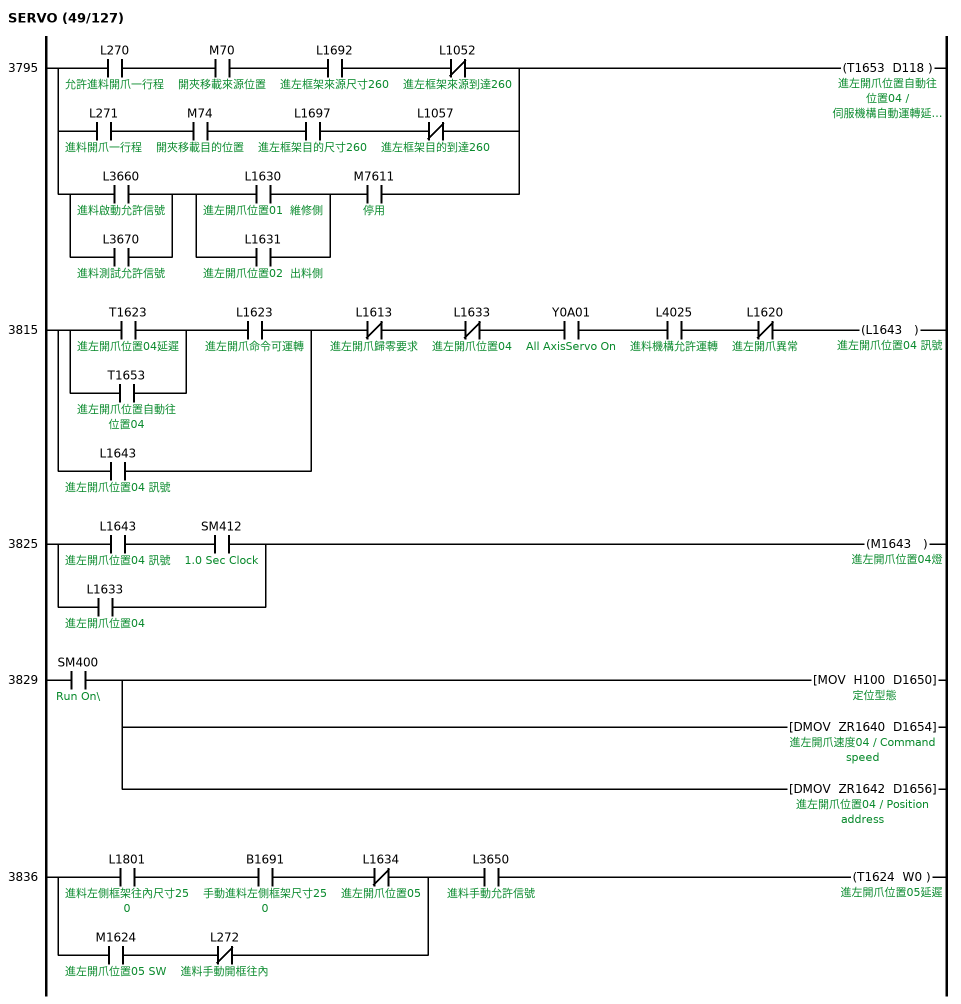
[picture p48: ladder of SERVO, rungs at steps 3795 to 3836]
3795  LD      L270  ; 允許進料開爪一行程
      AND     M70  ; 開夾移載來源位置
      AND     L1692  ; 進左框架來源尺寸260
      ANI     L1052  ; 進左框架來源到達260
      LD      L271  ; 進料開爪一行程
      AND     M74  ; 開夾移載目的位置
      AND     L1697  ; 進左框架目的尺寸260
      ANI     L1057  ; 進左框架目的到達260
      ORB
      LD      L3660  ; 進料啟動允許信號
      OR      L3670  ; 進料測試允許信號
      LD      L1630  ; 進左開爪位置01  維修側
      OR      L1631  ; 進左開爪位置02  出料側
      ANB
      AND     M7611  ; 停用
      ORB
      OUT     T1653 D118  ; 進左開爪位置自動往  位置04 / 伺服機構自動運轉延遲時間
3815  LD      T1623  ; 進左開爪位置04延遲
      OR      T1653  ; 進左開爪位置自動往  位置04
      AND     L1623  ; 進左開爪命令可運轉
      OR      L1643  ; 進左開爪位置04 訊號
      ANI     L1613  ; 進左開爪歸零要求
      ANI     L1633  ; 進左開爪位置04
      AND     Y0A01  ; All AxisServo On
      AND     L4025  ; 進料機構允許運轉
      ANI     L1620  ; 進左開爪異常
      OUT     L1643  ; 進左開爪位置04 訊號
3825  LD      L1643  ; 進左開爪位置04 訊號
      AND     SM412  ; 1.0 Sec Clock
      OR      L1633  ; 進左開爪位置04
      OUT     M1643  ; 進左開爪位置04燈
3829  LD      SM400  ; Run On\
      MOV     H100 D1650  ; 定位型態
      DMOV    ZR1640 D1654  ; 進左開爪速度04 / Command  speed
      DMOV    ZR1642 D1656  ; Position address
3836  LD      L1801  ; 進料左側框架往內尺寸250
      AND     B1691  ; 手動進料左側框架尺寸250
      ANI     L1634  ; 進左開爪位置05
      LD      M1624  ; 進左開爪位置05 SW
      ANI     L272  ; 進料手動開框往內
      ORB
      AND     L3650  ; 進料手動允許信號
      OUT     T1624 W0  ; 進左開爪位置05延遲
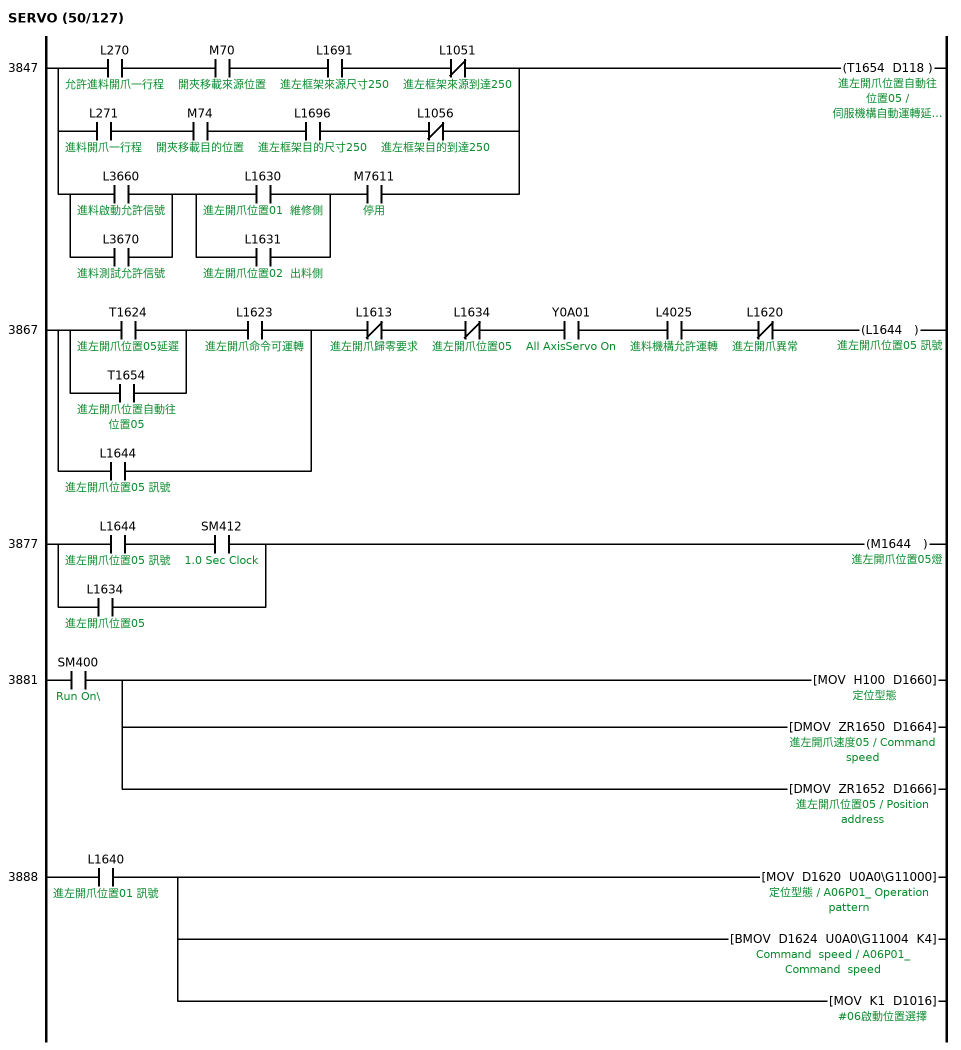
3847  LD      L270  ; 允許進料開爪一行程
      AND     M70  ; 開夾移載來源位置
      AND     L1691  ; 進左框架來源尺寸250
      ANI     L1051  ; 進左框架來源到達250
      LD      L271  ; 進料開爪一行程
      AND     M74  ; 開夾移載目的位置
      AND     L1696  ; 進左框架目的尺寸250
      ANI     L1056  ; 進左框架目的到達250
      ORB
      LD      L3660  ; 進料啟動允許信號
      OR      L3670  ; 進料測試允許信號
      LD      L1630  ; 進左開爪位置01  維修側
      OR      L1631  ; 進左開爪位置02  出料側
      ANB
      AND     M7611  ; 停用
      ORB
      OUT     T1654 D118  ; 進左開爪位置自動往  位置05 / 伺服機構自動運轉延遲時間
3867  LD      T1624  ; 進左開爪位置05延遲
      OR      T1654  ; 進左開爪位置自動往  位置05
      AND     L1623  ; 進左開爪命令可運轉
      OR      L1644  ; 進左開爪位置05 訊號
      ANI     L1613  ; 進左開爪歸零要求
      ANI     L1634  ; 進左開爪位置05
      AND     Y0A01  ; All AxisServo On
      AND     L4025  ; 進料機構允許運轉
      ANI     L1620  ; 進左開爪異常
      OUT     L1644  ; 進左開爪位置05 訊號
3877  LD      L1644  ; 進左開爪位置05 訊號
      AND     SM412  ; 1.0 Sec Clock
      OR      L1634  ; 進左開爪位置05
      OUT     M1644  ; 進左開爪位置05燈
3881  LD      SM400  ; Run On\
      MOV     H100 D1660  ; 定位型態
      DMOV    ZR1650 D1664  ; 進左開爪速度05 / Command  speed
      DMOV    ZR1652 D1666  ; Position address
3888  LD      L1640  ; 進左開爪位置01 訊號
      MOV     D1620 U0A0\G11000  ; A06P01_ Operation pattern
      BMOV    D1624 U0A0\G11004 K4  ; A06P01_ Command  speed
      MOV     K1 D1016  ; #06啟動位置選擇
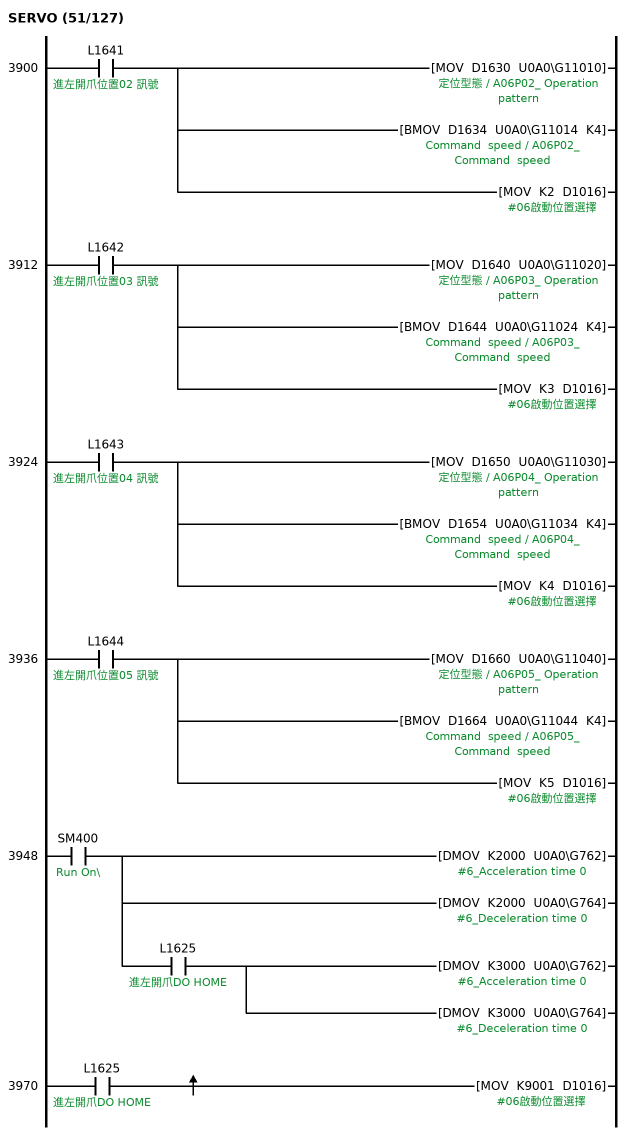
3900  LD      L1641  ; 進左開爪位置02 訊號
      MOV     D1630 U0A0\G11010  ; A06P02_ Operation pattern
      BMOV    D1634 U0A0\G11014 K4  ; A06P02_ Command  speed
      MOV     K2 D1016
3912  LD      L1642  ; 進左開爪位置03 訊號
      MOV     D1640 U0A0\G11020  ; A06P03_ Operation pattern
      BMOV    D1644 U0A0\G11024 K4  ; A06P03_ Command  speed
      MOV     K3 D1016
3924  LD      L1643  ; 進左開爪位置04 訊號
      MOV     D1650 U0A0\G11030  ; A06P04_ Operation pattern
      BMOV    D1654 U0A0\G11034 K4  ; A06P04_ Command  speed
      MOV     K4 D1016
3936  LD      L1644  ; 進左開爪位置05 訊號
      MOV     D1660 U0A0\G11040  ; A06P05_ Operation pattern
      BMOV    D1664 U0A0\G11044 K4  ; A06P05_ Command  speed
      MOV     K5 D1016
3948  LD      SM400  ; Run On\
      DMOV    K2000 U0A0\G762  ; #6_Acceleration time 0
      DMOV    K2000 U0A0\G764  ; #6_Deceleration time 0
      AND     L1625  ; 進左開爪DO HOME
      DMOV    K3000 U0A0\G762
      DMOV    K3000 U0A0\G764
3970  LD      L1625  ; 進左開爪DO HOME
      MEP
      MOV     K9001 D1016
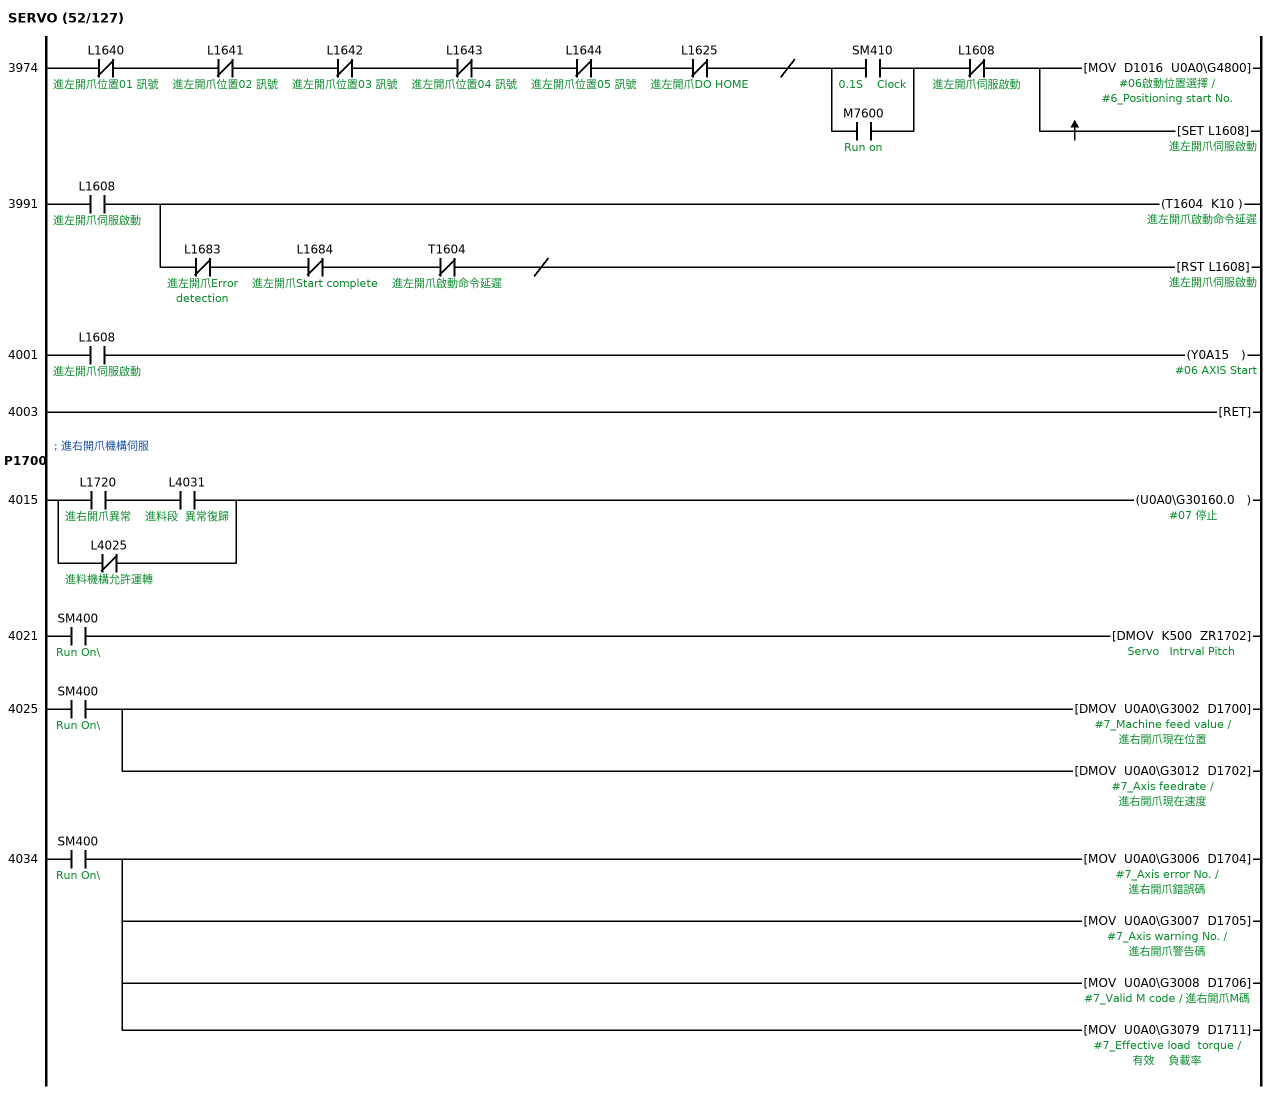
3974  LDI     L1640  ; 進左開爪位置01 訊號
      ANI     L1641  ; 進左開爪位置02 訊號
      ANI     L1642  ; 進左開爪位置03 訊號
      ANI     L1643  ; 進左開爪位置04 訊號
      ANI     L1644  ; 進左開爪位置05 訊號
      ANI     L1625  ; 進左開爪DO HOME
      INV
      LD      SM410  ; 0.1S    Clock
      OR      M7600  ; Run on
      ANB
      ANI     L1608  ; 進左開爪伺服啟動
      MOV     D1016 U0A0\G4800  ; #6_Positioning start No.
      MEP
      SET     L1608  ; 進左開爪伺服啟動
3991  LD      L1608  ; 進左開爪伺服啟動
      OUT     T1604 K10  ; 進左開爪啟動命令延遲
      ANI     L1683  ; 進左開爪Error detection
      ANI     L1684  ; 進左開爪Start complete
      ANI     T1604  ; 進左開爪啟動命令延遲
      INV
      RST     L1608  ; 進左開爪伺服啟動
4001  LD      L1608  ; 進左開爪伺服啟動
      OUT     Y0A15  ; #06 AXIS Start
4003  RET
; 進右開爪機構伺服
      P1700
4015  LD      L1720  ; 進右開爪異常
      AND     L4031  ; 進料段  異常復歸
      ORI     L4025  ; 進料機構允許運轉
      OUT     U0A0\G30160.0  ; #07 停止
4021  LD      SM400  ; Run On\
      DMOV    K500 ZR1702  ; Servo   Intrval Pitch
4025  LD      SM400  ; Run On\
      DMOV    U0A0\G3002 D1700  ; #7_Machine feed value / 進右開爪現在位置
      DMOV    U0A0\G3012 D1702  ; #7_Axis feedrate / 進右開爪現在速度
4034  LD      SM400  ; Run On\
      MOV     U0A0\G3006 D1704  ; #7_Axis error No. / 進右開爪錯誤碼
      MOV     U0A0\G3007 D1705  ; #7_Axis warning No. / 進右開爪警告碼
      MOV     U0A0\G3008 D1706  ; #7_Valid M code / 進右開爪M碼
      MOV     U0A0\G3079 D1711  ; #7_Effective load  torque / 有效    負載率
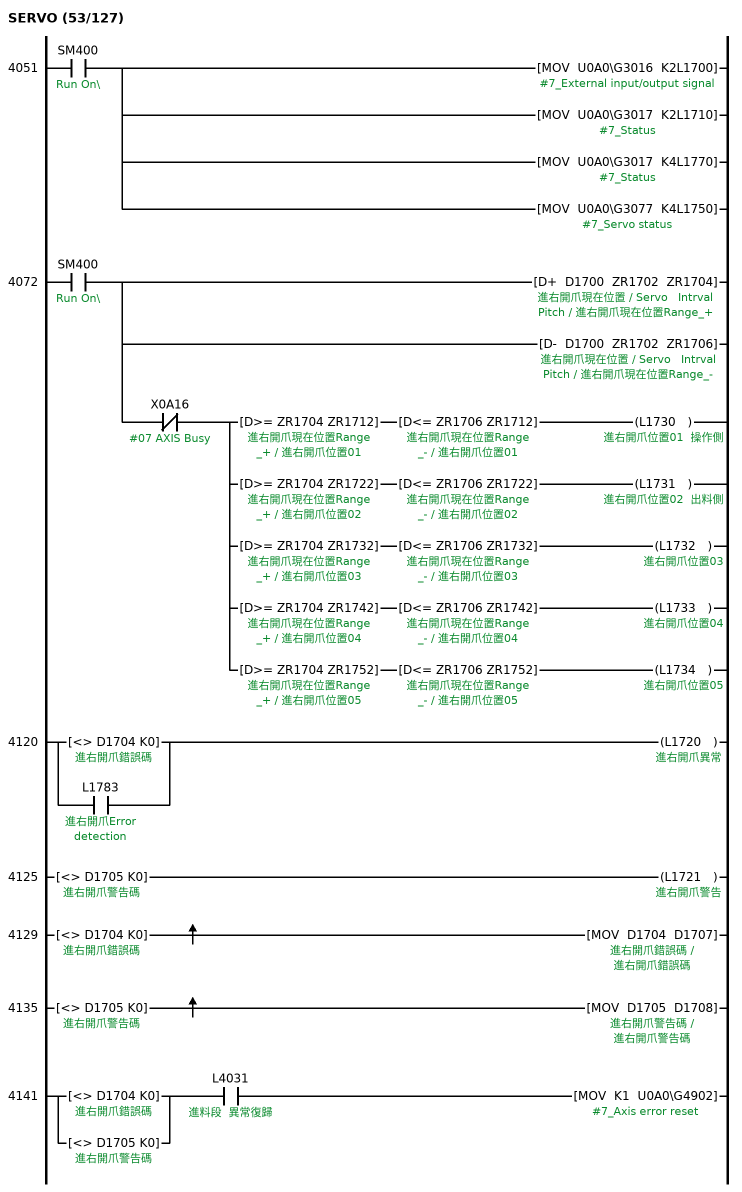
4051  LD      SM400  ; Run On\
      MOV     U0A0\G3016 K2L1700  ; #7_External input/output signal / 進右開爪  負極限
      MOV     U0A0\G3017 K2L1710  ; #7_Status / 進右開爪速度控制
      MOV     U0A0\G3017 K4L1770  ; 進右開爪速度控制
      MOV     U0A0\G3077 K4L1750  ; #7_Servo status / READY ON
4072  LD      SM400  ; Run On\
      D+      D1700 ZR1702 ZR1704  ; 進右開爪現在位置Range_+
      D-      D1700 ZR1702 ZR1706  ; 進右開爪現在位置Range_-
      ANI     X0A16  ; #07 AXIS Busy
      MPS
      ANDD>=  ZR1704 ZR1712  ; 進右開爪現在位置Range_+ / 進右開爪位置01
      ANDD<=  ZR1706 ZR1712  ; 進右開爪現在位置Range_- / 進右開爪位置01
      OUT     L1730  ; 進右開爪位置01  操作側
      MRD
      ANDD>=  ZR1704 ZR1722  ; 進右開爪現在位置Range_+ / 進右開爪位置02
      ANDD<=  ZR1706 ZR1722  ; 進右開爪現在位置Range_- / 進右開爪位置02
      OUT     L1731  ; 進右開爪位置02  出料側
      MRD
      ANDD>=  ZR1704 ZR1732  ; 進右開爪現在位置Range_+ / 進右開爪位置03
      ANDD<=  ZR1706 ZR1732  ; 進右開爪現在位置Range_- / 進右開爪位置03
      OUT     L1732  ; 進右開爪位置03
      MRD
      ANDD>=  ZR1704 ZR1742  ; 進右開爪現在位置Range_+ / 進右開爪位置04
      ANDD<=  ZR1706 ZR1742  ; 進右開爪現在位置Range_- / 進右開爪位置04
      OUT     L1733  ; 進右開爪位置04
      MPP
      ANDD>=  ZR1704 ZR1752  ; 進右開爪現在位置Range_+ / 進右開爪位置05
      ANDD<=  ZR1706 ZR1752  ; 進右開爪現在位置Range_- / 進右開爪位置05
      OUT     L1734  ; 進右開爪位置05
4120  LD<>    D1704 K0  ; 進右開爪錯誤碼
      OR      L1783  ; 進右開爪Error detection
      OUT     L1720  ; 進右開爪異常
4125  LD<>    D1705 K0  ; 進右開爪警告碼
      OUT     L1721  ; 進右開爪警告
4129  LD<>    D1704 K0  ; 進右開爪錯誤碼
      MEP
      MOV     D1704 D1707  ; 進右開爪錯誤碼
4135  LD<>    D1705 K0  ; 進右開爪警告碼
      MEP
      MOV     D1705 D1708  ; 進右開爪警告碼
4141  LD<>    D1704 K0  ; 進右開爪錯誤碼
      OR<>    D1705 K0  ; 進右開爪警告碼
      AND     L4031  ; 進料段  異常復歸
      MOV     K1 U0A0\G4902  ; #7_Axis error reset
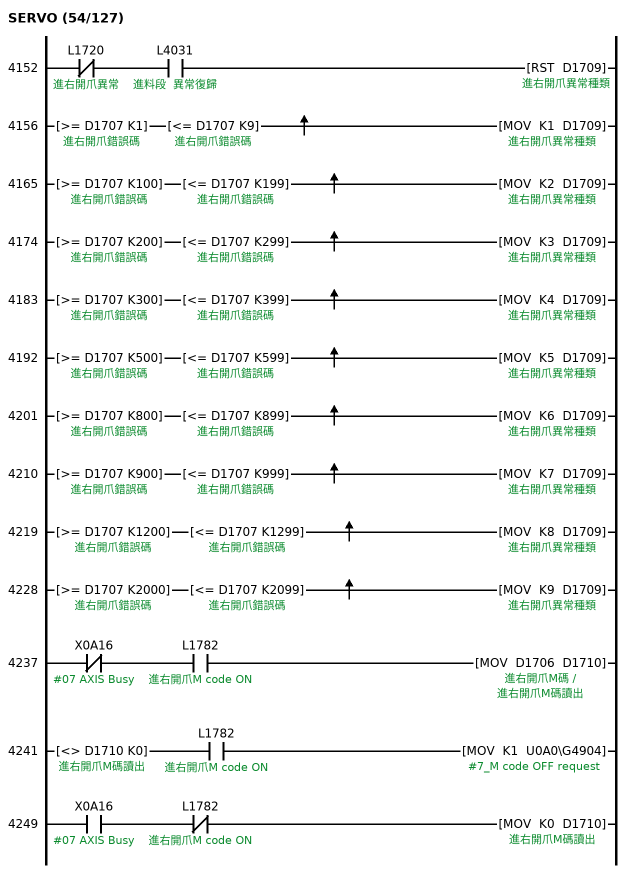
4152  LDI     L1720  ; 進右開爪異常
      AND     L4031  ; 進料段  異常復歸
      RST     D1709  ; 進右開爪異常種類
4156  LD>=    D1707 K1  ; 進右開爪錯誤碼
      AND<=   D1707 K9  ; 進右開爪錯誤碼
      MEP
      MOV     K1 D1709
4165  LD>=    D1707 K100  ; 進右開爪錯誤碼
      AND<=   D1707 K199  ; 進右開爪錯誤碼
      MEP
      MOV     K2 D1709
4174  LD>=    D1707 K200  ; 進右開爪錯誤碼
      AND<=   D1707 K299  ; 進右開爪錯誤碼
      MEP
      MOV     K3 D1709
4183  LD>=    D1707 K300  ; 進右開爪錯誤碼
      AND<=   D1707 K399  ; 進右開爪錯誤碼
      MEP
      MOV     K4 D1709
4192  LD>=    D1707 K500  ; 進右開爪錯誤碼
      AND<=   D1707 K599  ; 進右開爪錯誤碼
      MEP
      MOV     K5 D1709
4201  LD>=    D1707 K800  ; 進右開爪錯誤碼
      AND<=   D1707 K899  ; 進右開爪錯誤碼
      MEP
      MOV     K6 D1709
4210  LD>=    D1707 K900  ; 進右開爪錯誤碼
      AND<=   D1707 K999  ; 進右開爪錯誤碼
      MEP
      MOV     K7 D1709
4219  LD>=    D1707 K1200  ; 進右開爪錯誤碼
      AND<=   D1707 K1299  ; 進右開爪錯誤碼
      MEP
      MOV     K8 D1709
4228  LD>=    D1707 K2000  ; 進右開爪錯誤碼
      AND<=   D1707 K2099  ; 進右開爪錯誤碼
      MEP
      MOV     K9 D1709
4237  LDI     X0A16  ; #07 AXIS Busy
      AND     L1782  ; 進右開爪M code ON
      MOV     D1706 D1710  ; 進右開爪M碼讀出
4241  LD<>    D1710 K0  ; 進右開爪M碼讀出
      AND     L1782  ; 進右開爪M code ON
      MOV     K1 U0A0\G4904  ; #7_M code OFF request
4249  LD      X0A16  ; #07 AXIS Busy
      ANI     L1782  ; 進右開爪M code ON
      MOV     K0 D1710
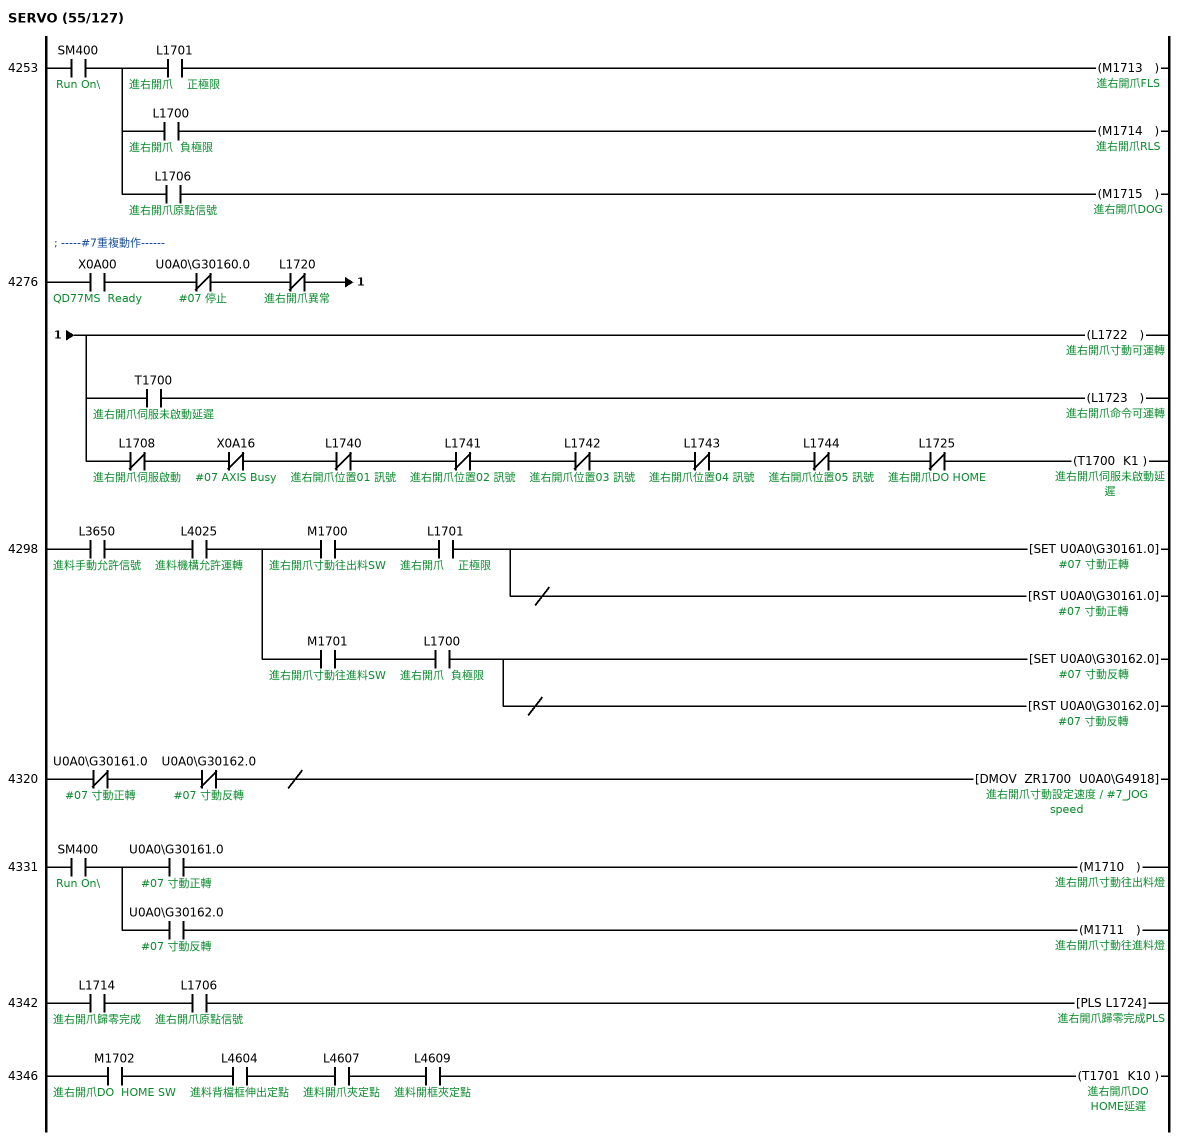
4253  LD      SM400  ; Run On\
      MPS
      AND     L1701  ; 進右開爪    正極限
      OUT     M1713  ; 進右開爪FLS
      MRD
      AND     L1700  ; 進右開爪  負極限
      OUT     M1714  ; 進右開爪RLS
      MPP
      AND     L1706  ; 進右開爪原點信號
      OUT     M1715  ; 進右開爪DOG
; -----#7重複動作------
4276  LD      X0A00  ; QD77MS  Ready
      ANI     U0A0\G30160.0  ; #07 停止
      ANI     L1720  ; 進右開爪異常
      OUT     L1722  ; 進右開爪寸動可運轉
      MPS
      AND     T1700  ; 進右開爪伺服未啟動延遲
      OUT     L1723  ; 進右開爪命令可運轉
      MPP
      ANI     L1708  ; 進右開爪伺服啟動
      ANI     X0A16  ; #07 AXIS Busy
      ANI     L1740  ; 進右開爪位置01 訊號
      ANI     L1741  ; 進右開爪位置02 訊號
      ANI     L1742  ; 進右開爪位置03 訊號
      ANI     L1743  ; 進右開爪位置04 訊號
      ANI     L1744  ; 進右開爪位置05 訊號
      ANI     L1725  ; 進右開爪DO HOME
      OUT     T1700 K1  ; 進右開爪伺服未啟動延遲
4298  LD      L3650  ; 進料手動允許信號
      AND     L4025  ; 進料機構允許運轉
      MPS
      AND     M1700  ; 進右開爪寸動往出料SW
      AND     L1701  ; 進右開爪    正極限
      SET     U0A0\G30161.0  ; #07 寸動正轉
      INV
      RST     U0A0\G30161.0  ; #07 寸動正轉
      MPP
      AND     M1701  ; 進右開爪寸動往進料SW
      AND     L1700  ; 進右開爪  負極限
      SET     U0A0\G30162.0  ; #07 寸動反轉
      INV
      RST     U0A0\G30162.0  ; #07 寸動反轉
4320  LDI     U0A0\G30161.0  ; #07 寸動正轉
      ANI     U0A0\G30162.0  ; #07 寸動反轉
      INV
      DMOV    ZR1700 U0A0\G4918  ; 進右開爪寸動設定速度 / #7_JOG     speed
4331  LD      SM400  ; Run On\
      MPS
      AND     U0A0\G30161.0  ; #07 寸動正轉
      OUT     M1710  ; 進右開爪寸動往出料燈
      MPP
      AND     U0A0\G30162.0  ; #07 寸動反轉
      OUT     M1711  ; 進右開爪寸動往進料燈
4342  LD      L1714  ; 進右開爪歸零完成
      AND     L1706  ; 進右開爪原點信號
      PLS     L1724  ; 進右開爪歸零完成PLS
4346  LD      M1702  ; 進右開爪DO  HOME SW
      AND     L4604  ; 進料背檔框伸出定點
      AND     L4607  ; 進料開爪夾定點
      AND     L4609  ; 進料開框夾定點
      OUT     T1701 K10  ; 進右開爪DO HOME延遲
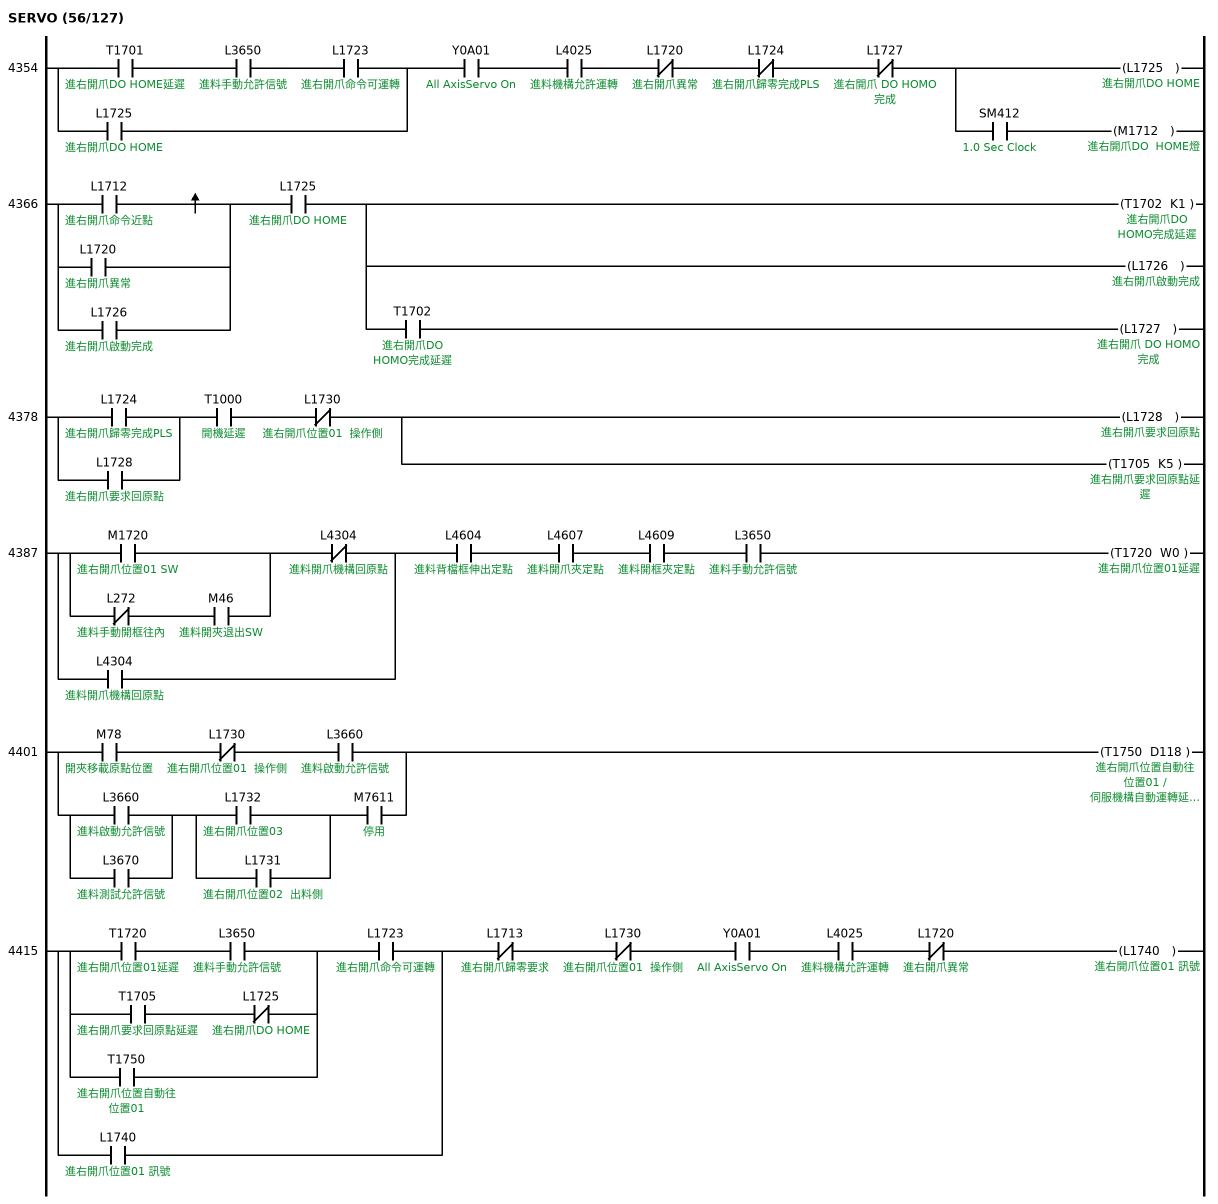
4354  LD      T1701  ; 進右開爪DO HOME延遲
      AND     L3650  ; 進料手動允許信號
      AND     L1723  ; 進右開爪命令可運轉
      OR      L1725  ; 進右開爪DO HOME
      AND     Y0A01  ; All AxisServo On
      AND     L4025  ; 進料機構允許運轉
      ANI     L1720  ; 進右開爪異常
      ANI     L1724  ; 進右開爪歸零完成PLS
      ANI     L1727  ; 進右開爪 DO HOMO 完成
      OUT     L1725  ; 進右開爪DO HOME
      AND     SM412  ; 1.0 Sec Clock
      OUT     M1712  ; 進右開爪DO  HOME燈
4366  LD      L1712  ; 進右開爪命令近點
      MEP
      OR      L1720  ; 進右開爪異常
      OR      L1726  ; 進右開爪啟動完成
      AND     L1725  ; 進右開爪DO HOME
      OUT     T1702 K1  ; 進右開爪DO HOMO完成延遲
      OUT     L1726  ; 進右開爪啟動完成
      AND     T1702  ; 進右開爪DO HOMO完成延遲
      OUT     L1727  ; 進右開爪 DO HOMO 完成
4378  LD      L1724  ; 進右開爪歸零完成PLS
      OR      L1728  ; 進右開爪要求回原點
      AND     T1000  ; 開機延遲
      ANI     L1730  ; 進右開爪位置01  操作側
      OUT     L1728  ; 進右開爪要求回原點
      OUT     T1705 K5  ; 進右開爪要求回原點延遲
4387  LD      M1720  ; 進右開爪位置01 SW
      LDI     L272  ; 進料手動開框往內
      AND     M46  ; 進料開夾退出SW
      ORB
      ANI     L4304  ; 進料開爪機構回原點
      OR      L4304  ; 進料開爪機構回原點
      AND     L4604  ; 進料背檔框伸出定點
      AND     L4607  ; 進料開爪夾定點
      AND     L4609  ; 進料開框夾定點
      AND     L3650  ; 進料手動允許信號
      OUT     T1720 W0  ; 進右開爪位置01延遲
4401  LD      M78  ; 開夾移載原點位置
      ANI     L1730  ; 進右開爪位置01  操作側
      AND     L3660  ; 進料啟動允許信號
      LD      L3660  ; 進料啟動允許信號
      OR      L3670  ; 進料測試允許信號
      LD      L1732  ; 進右開爪位置03
      OR      L1731  ; 進右開爪位置02  出料側
      ANB
      AND     M7611  ; 停用
      ORB
      OUT     T1750 D118  ; 進右開爪位置自動往  位置01 / 伺服機構自動運轉延遲時間
4415  LD      T1720  ; 進右開爪位置01延遲
      AND     L3650  ; 進料手動允許信號
      LD      T1705  ; 進右開爪要求回原點延遲
      ANI     L1725  ; 進右開爪DO HOME
      ORB
      OR      T1750  ; 進右開爪位置自動往  位置01
      AND     L1723  ; 進右開爪命令可運轉
      OR      L1740  ; 進右開爪位置01 訊號
      ANI     L1713  ; 進右開爪歸零要求
      ANI     L1730  ; 進右開爪位置01  操作側
      AND     Y0A01  ; All AxisServo On
      AND     L4025  ; 進料機構允許運轉
      ANI     L1720  ; 進右開爪異常
      OUT     L1740  ; 進右開爪位置01 訊號
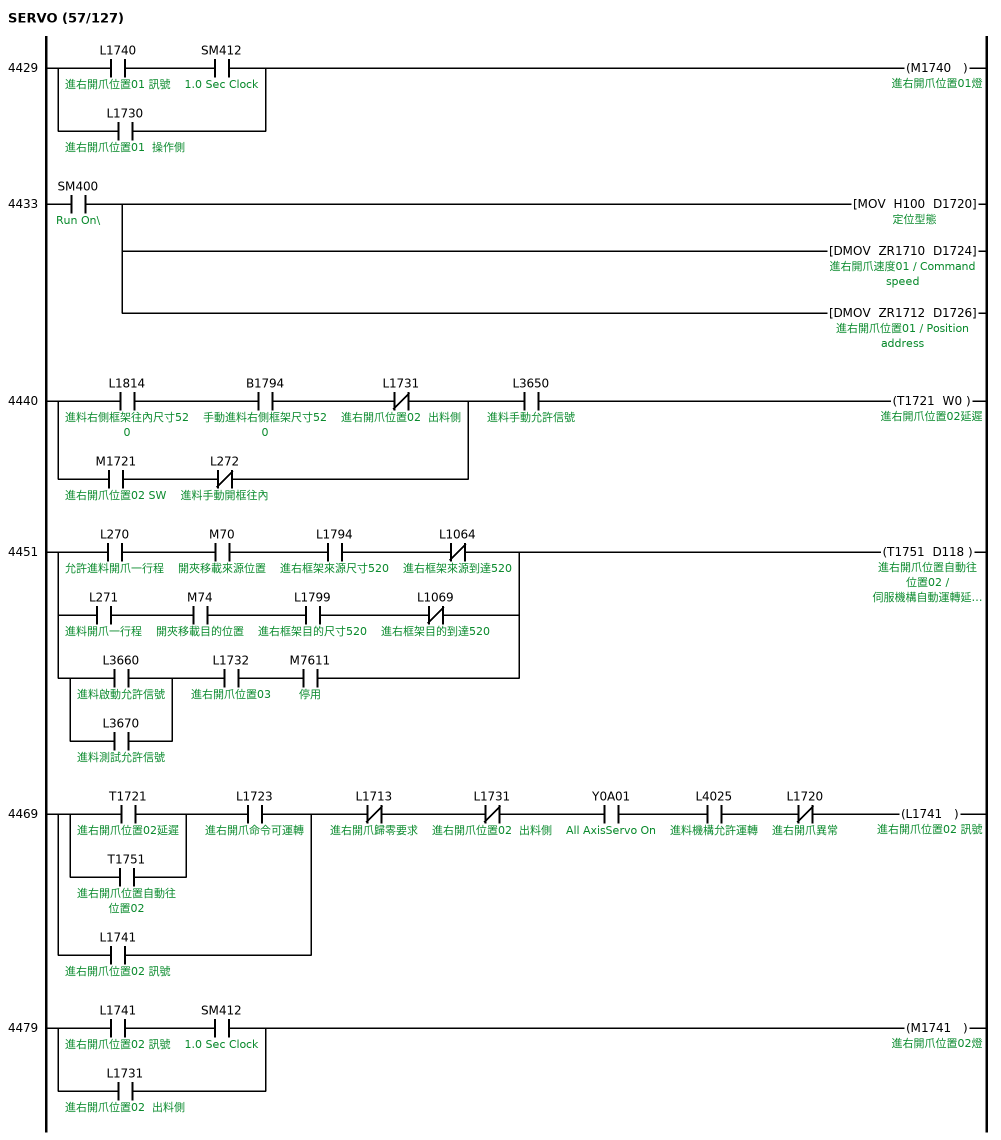
4429  LD      L1740  ; 進右開爪位置01 訊號
      AND     SM412  ; 1.0 Sec Clock
      OR      L1730  ; 進右開爪位置01  操作側
      OUT     M1740  ; 進右開爪位置01燈
4433  LD      SM400  ; Run On\
      MOV     H100 D1720  ; 定位型態
      DMOV    ZR1710 D1724  ; 進右開爪速度01 / Command  speed
      DMOV    ZR1712 D1726  ; Position address
4440  LD      L1814  ; 進料右側框架往內尺寸520
      AND     B1794  ; 手動進料右側框架尺寸520
      ANI     L1731  ; 進右開爪位置02  出料側
      LD      M1721  ; 進右開爪位置02 SW
      ANI     L272  ; 進料手動開框往內
      ORB
      AND     L3650  ; 進料手動允許信號
      OUT     T1721 W0  ; 進右開爪位置02延遲
4451  LD      L270  ; 允許進料開爪一行程
      AND     M70  ; 開夾移載來源位置
      AND     L1794  ; 進右框架來源尺寸520
      ANI     L1064  ; 進右框架來源到達520
      LD      L271  ; 進料開爪一行程
      AND     M74  ; 開夾移載目的位置
      AND     L1799  ; 進右框架目的尺寸520
      ANI     L1069  ; 進右框架目的到達520
      ORB
      LD      L3660  ; 進料啟動允許信號
      OR      L3670  ; 進料測試允許信號
      AND     L1732  ; 進右開爪位置03
      AND     M7611  ; 停用
      ORB
      OUT     T1751 D118  ; 進右開爪位置自動往  位置02 / 伺服機構自動運轉延遲時間
4469  LD      T1721  ; 進右開爪位置02延遲
      OR      T1751  ; 進右開爪位置自動往  位置02
      AND     L1723  ; 進右開爪命令可運轉
      OR      L1741  ; 進右開爪位置02 訊號
      ANI     L1713  ; 進右開爪歸零要求
      ANI     L1731  ; 進右開爪位置02  出料側
      AND     Y0A01  ; All AxisServo On
      AND     L4025  ; 進料機構允許運轉
      ANI     L1720  ; 進右開爪異常
      OUT     L1741  ; 進右開爪位置02 訊號
4479  LD      L1741  ; 進右開爪位置02 訊號
      AND     SM412  ; 1.0 Sec Clock
      OR      L1731  ; 進右開爪位置02  出料側
      OUT     M1741  ; 進右開爪位置02燈
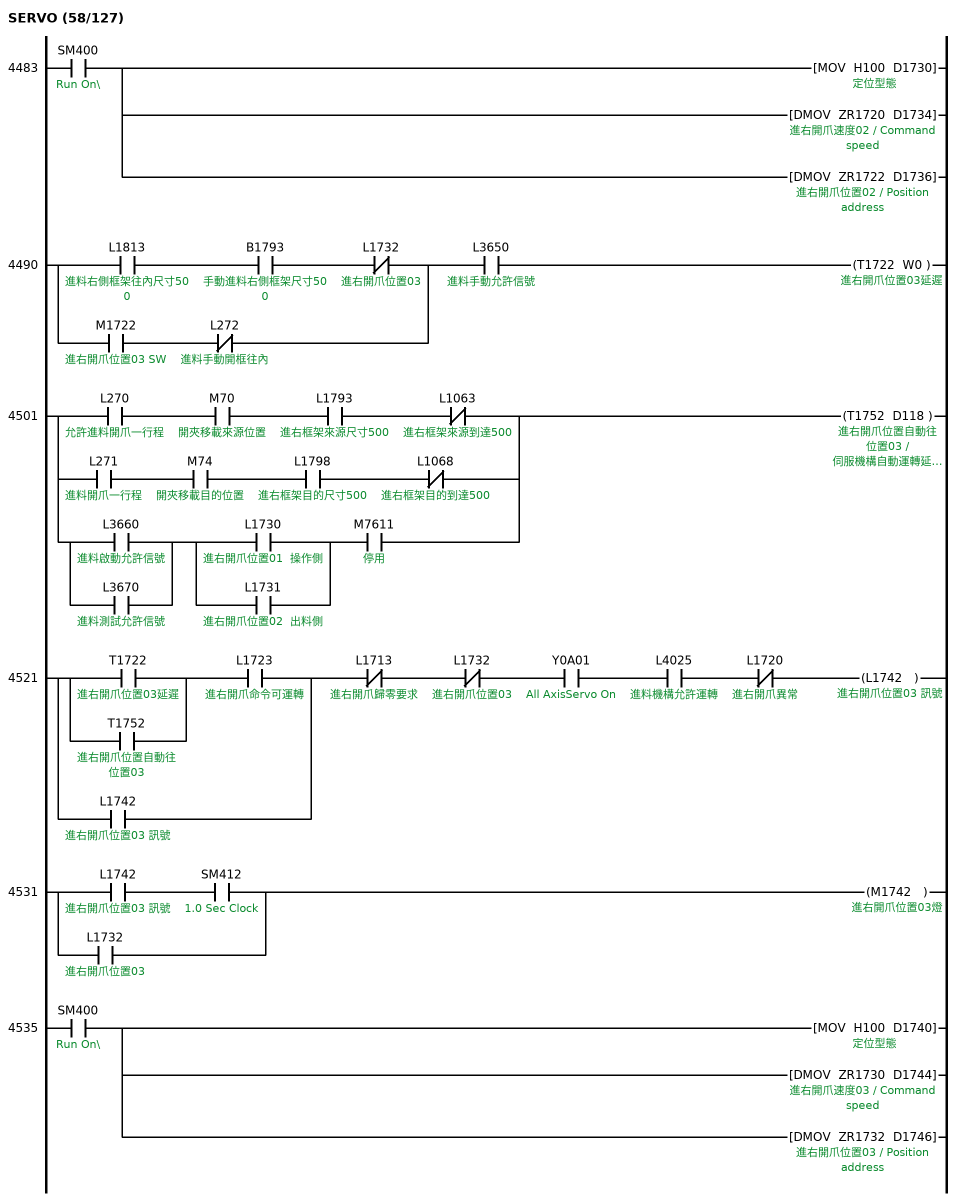
4483  LD      SM400  ; Run On\
      MOV     H100 D1730  ; 定位型態
      DMOV    ZR1720 D1734  ; 進右開爪速度02 / Command  speed
      DMOV    ZR1722 D1736  ; Position address
4490  LD      L1813  ; 進料右側框架往內尺寸500
      AND     B1793  ; 手動進料右側框架尺寸500
      ANI     L1732  ; 進右開爪位置03
      LD      M1722  ; 進右開爪位置03 SW
      ANI     L272  ; 進料手動開框往內
      ORB
      AND     L3650  ; 進料手動允許信號
      OUT     T1722 W0  ; 進右開爪位置03延遲
4501  LD      L270  ; 允許進料開爪一行程
      AND     M70  ; 開夾移載來源位置
      AND     L1793  ; 進右框架來源尺寸500
      ANI     L1063  ; 進右框架來源到達500
      LD      L271  ; 進料開爪一行程
      AND     M74  ; 開夾移載目的位置
      AND     L1798  ; 進右框架目的尺寸500
      ANI     L1068  ; 進右框架目的到達500
      ORB
      LD      L3660  ; 進料啟動允許信號
      OR      L3670  ; 進料測試允許信號
      LD      L1730  ; 進右開爪位置01  操作側
      OR      L1731  ; 進右開爪位置02  出料側
      ANB
      AND     M7611  ; 停用
      ORB
      OUT     T1752 D118  ; 進右開爪位置自動往  位置03 / 伺服機構自動運轉延遲時間
4521  LD      T1722  ; 進右開爪位置03延遲
      OR      T1752  ; 進右開爪位置自動往  位置03
      AND     L1723  ; 進右開爪命令可運轉
      OR      L1742  ; 進右開爪位置03 訊號
      ANI     L1713  ; 進右開爪歸零要求
      ANI     L1732  ; 進右開爪位置03
      AND     Y0A01  ; All AxisServo On
      AND     L4025  ; 進料機構允許運轉
      ANI     L1720  ; 進右開爪異常
      OUT     L1742  ; 進右開爪位置03 訊號
4531  LD      L1742  ; 進右開爪位置03 訊號
      AND     SM412  ; 1.0 Sec Clock
      OR      L1732  ; 進右開爪位置03
      OUT     M1742  ; 進右開爪位置03燈
4535  LD      SM400  ; Run On\
      MOV     H100 D1740  ; 定位型態
      DMOV    ZR1730 D1744  ; 進右開爪速度03 / Command  speed
      DMOV    ZR1732 D1746  ; Position address
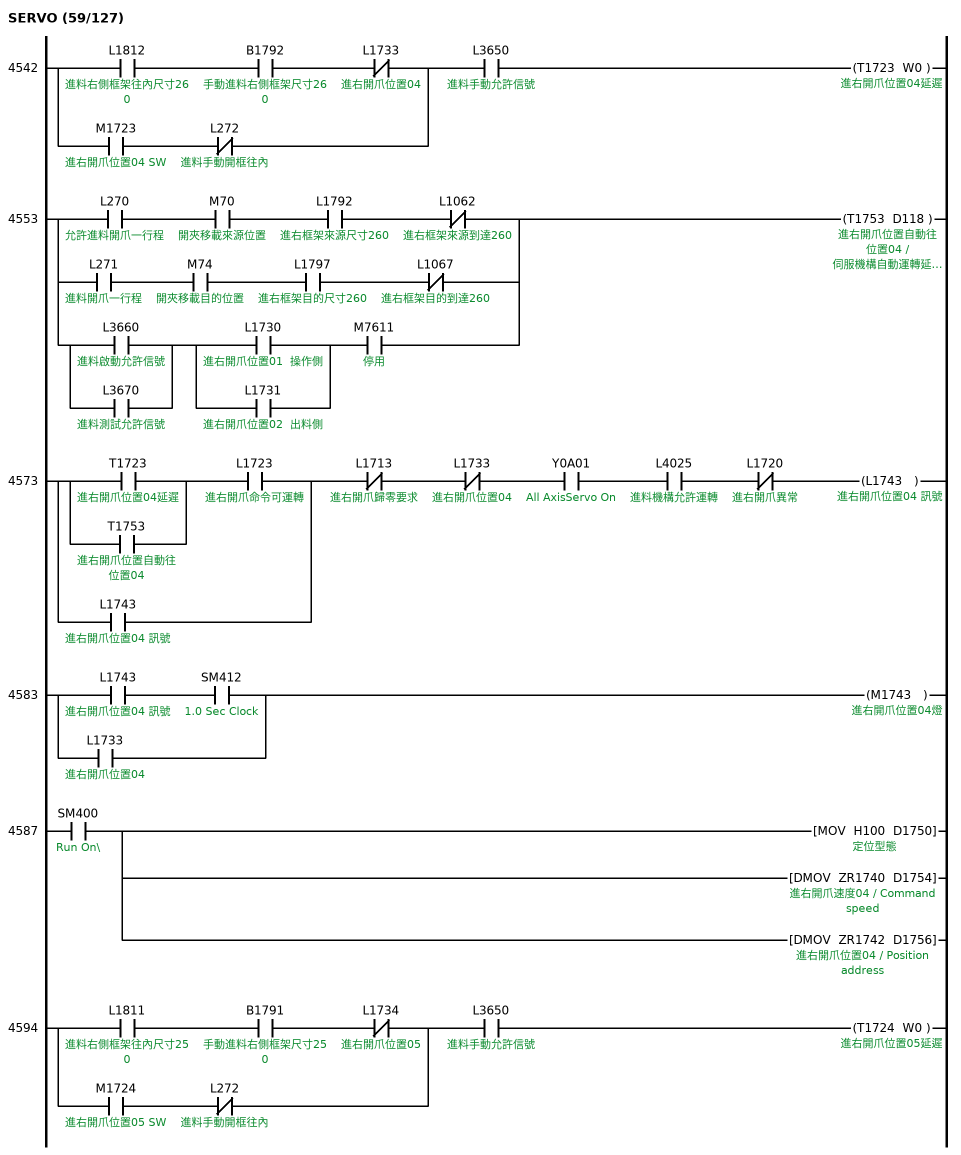
4542  LD      L1812  ; 進料右側框架往內尺寸260
      AND     B1792  ; 手動進料右側框架尺寸260
      ANI     L1733  ; 進右開爪位置04
      LD      M1723  ; 進右開爪位置04 SW
      ANI     L272  ; 進料手動開框往內
      ORB
      AND     L3650  ; 進料手動允許信號
      OUT     T1723 W0  ; 進右開爪位置04延遲
4553  LD      L270  ; 允許進料開爪一行程
      AND     M70  ; 開夾移載來源位置
      AND     L1792  ; 進右框架來源尺寸260
      ANI     L1062  ; 進右框架來源到達260
      LD      L271  ; 進料開爪一行程
      AND     M74  ; 開夾移載目的位置
      AND     L1797  ; 進右框架目的尺寸260
      ANI     L1067  ; 進右框架目的到達260
      ORB
      LD      L3660  ; 進料啟動允許信號
      OR      L3670  ; 進料測試允許信號
      LD      L1730  ; 進右開爪位置01  操作側
      OR      L1731  ; 進右開爪位置02  出料側
      ANB
      AND     M7611  ; 停用
      ORB
      OUT     T1753 D118  ; 進右開爪位置自動往  位置04 / 伺服機構自動運轉延遲時間
4573  LD      T1723  ; 進右開爪位置04延遲
      OR      T1753  ; 進右開爪位置自動往  位置04
      AND     L1723  ; 進右開爪命令可運轉
      OR      L1743  ; 進右開爪位置04 訊號
      ANI     L1713  ; 進右開爪歸零要求
      ANI     L1733  ; 進右開爪位置04
      AND     Y0A01  ; All AxisServo On
      AND     L4025  ; 進料機構允許運轉
      ANI     L1720  ; 進右開爪異常
      OUT     L1743  ; 進右開爪位置04 訊號
4583  LD      L1743  ; 進右開爪位置04 訊號
      AND     SM412  ; 1.0 Sec Clock
      OR      L1733  ; 進右開爪位置04
      OUT     M1743  ; 進右開爪位置04燈
4587  LD      SM400  ; Run On\
      MOV     H100 D1750  ; 定位型態
      DMOV    ZR1740 D1754  ; 進右開爪速度04 / Command  speed
      DMOV    ZR1742 D1756  ; Position address
4594  LD      L1811  ; 進料右側框架往內尺寸250
      AND     B1791  ; 手動進料右側框架尺寸250
      ANI     L1734  ; 進右開爪位置05
      LD      M1724  ; 進右開爪位置05 SW
      ANI     L272  ; 進料手動開框往內
      ORB
      AND     L3650  ; 進料手動允許信號
      OUT     T1724 W0  ; 進右開爪位置05延遲
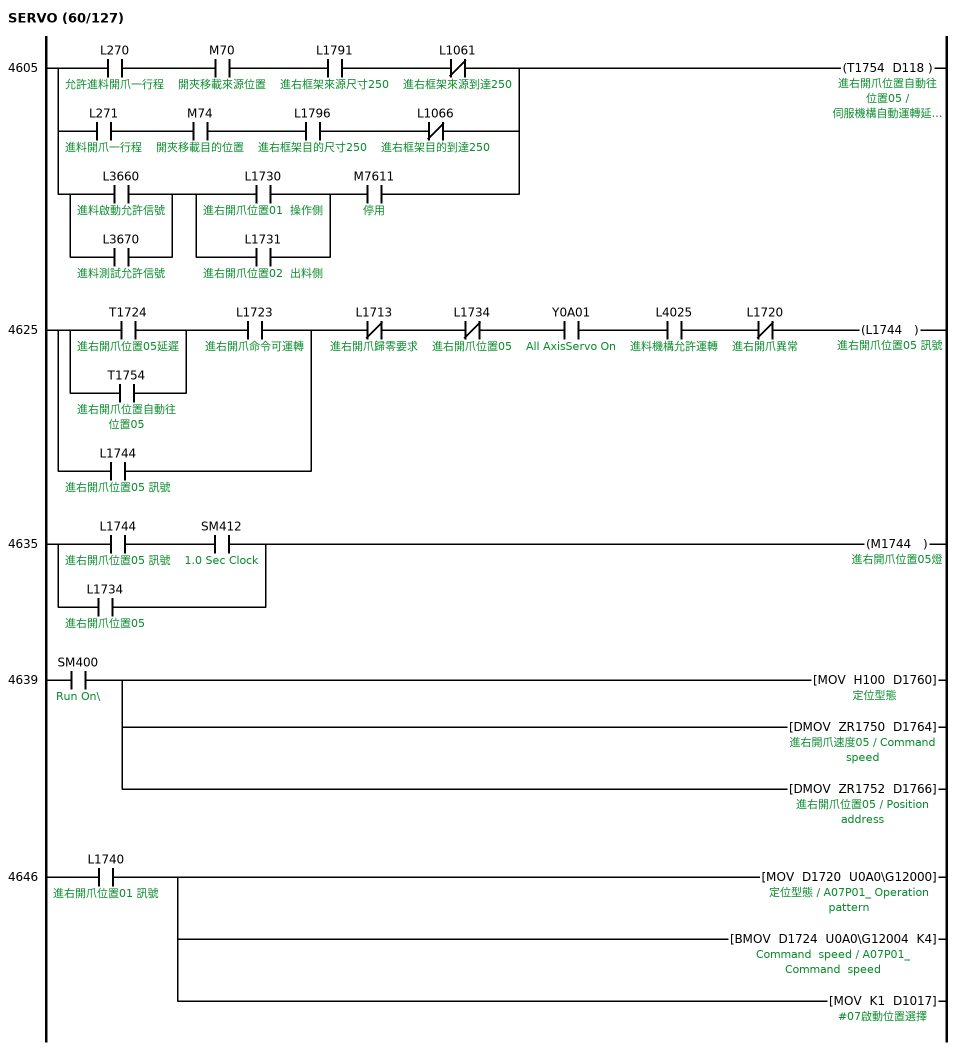
4605  LD      L270  ; 允許進料開爪一行程
      AND     M70  ; 開夾移載來源位置
      AND     L1791  ; 進右框架來源尺寸250
      ANI     L1061  ; 進右框架來源到達250
      LD      L271  ; 進料開爪一行程
      AND     M74  ; 開夾移載目的位置
      AND     L1796  ; 進右框架目的尺寸250
      ANI     L1066  ; 進右框架目的到達250
      ORB
      LD      L3660  ; 進料啟動允許信號
      OR      L3670  ; 進料測試允許信號
      LD      L1730  ; 進右開爪位置01  操作側
      OR      L1731  ; 進右開爪位置02  出料側
      ANB
      AND     M7611  ; 停用
      ORB
      OUT     T1754 D118  ; 進右開爪位置自動往  位置05 / 伺服機構自動運轉延遲時間
4625  LD      T1724  ; 進右開爪位置05延遲
      OR      T1754  ; 進右開爪位置自動往  位置05
      AND     L1723  ; 進右開爪命令可運轉
      OR      L1744  ; 進右開爪位置05 訊號
      ANI     L1713  ; 進右開爪歸零要求
      ANI     L1734  ; 進右開爪位置05
      AND     Y0A01  ; All AxisServo On
      AND     L4025  ; 進料機構允許運轉
      ANI     L1720  ; 進右開爪異常
      OUT     L1744  ; 進右開爪位置05 訊號
4635  LD      L1744  ; 進右開爪位置05 訊號
      AND     SM412  ; 1.0 Sec Clock
      OR      L1734  ; 進右開爪位置05
      OUT     M1744  ; 進右開爪位置05燈
4639  LD      SM400  ; Run On\
      MOV     H100 D1760  ; 定位型態
      DMOV    ZR1750 D1764  ; 進右開爪速度05 / Command  speed
      DMOV    ZR1752 D1766  ; Position address
4646  LD      L1740  ; 進右開爪位置01 訊號
      MOV     D1720 U0A0\G12000  ; A07P01_ Operation pattern
      BMOV    D1724 U0A0\G12004 K4  ; A07P01_ Command  speed
      MOV     K1 D1017  ; #07啟動位置選擇
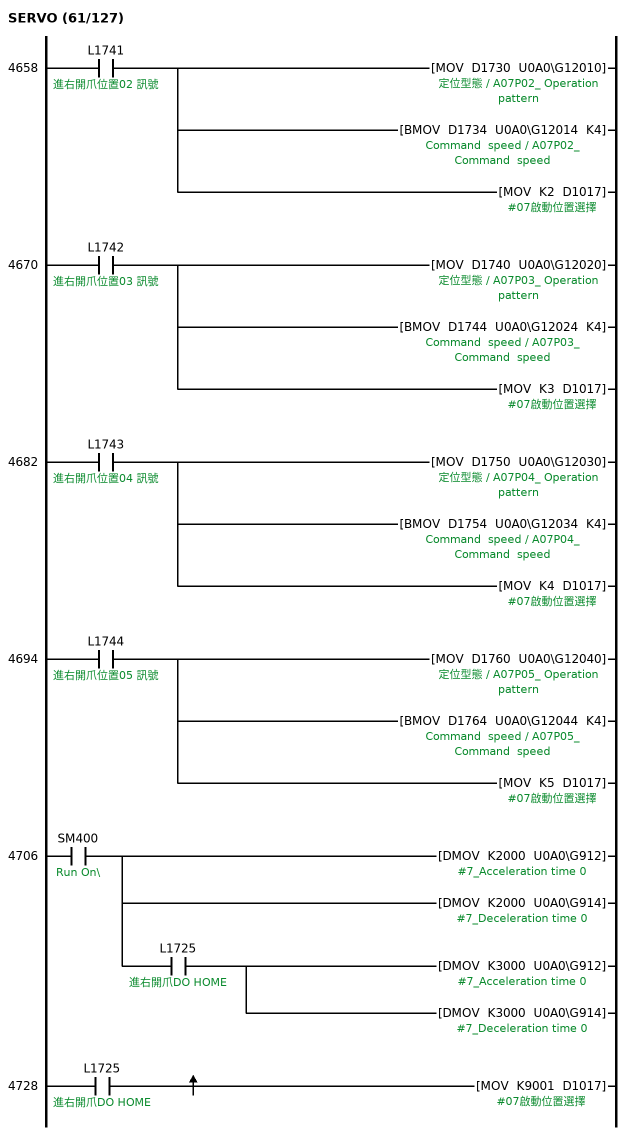
4658  LD      L1741  ; 進右開爪位置02 訊號
      MOV     D1730 U0A0\G12010  ; A07P02_ Operation pattern
      BMOV    D1734 U0A0\G12014 K4  ; A07P02_ Command  speed
      MOV     K2 D1017
4670  LD      L1742  ; 進右開爪位置03 訊號
      MOV     D1740 U0A0\G12020  ; A07P03_ Operation pattern
      BMOV    D1744 U0A0\G12024 K4  ; A07P03_ Command  speed
      MOV     K3 D1017
4682  LD      L1743  ; 進右開爪位置04 訊號
      MOV     D1750 U0A0\G12030  ; A07P04_ Operation pattern
      BMOV    D1754 U0A0\G12034 K4  ; A07P04_ Command  speed
      MOV     K4 D1017
4694  LD      L1744  ; 進右開爪位置05 訊號
      MOV     D1760 U0A0\G12040  ; A07P05_ Operation pattern
      BMOV    D1764 U0A0\G12044 K4  ; A07P05_ Command  speed
      MOV     K5 D1017
4706  LD      SM400  ; Run On\
      DMOV    K2000 U0A0\G912  ; #7_Acceleration time 0
      DMOV    K2000 U0A0\G914  ; #7_Deceleration time 0
      AND     L1725  ; 進右開爪DO HOME
      DMOV    K3000 U0A0\G912
      DMOV    K3000 U0A0\G914
4728  LD      L1725  ; 進右開爪DO HOME
      MEP
      MOV     K9001 D1017
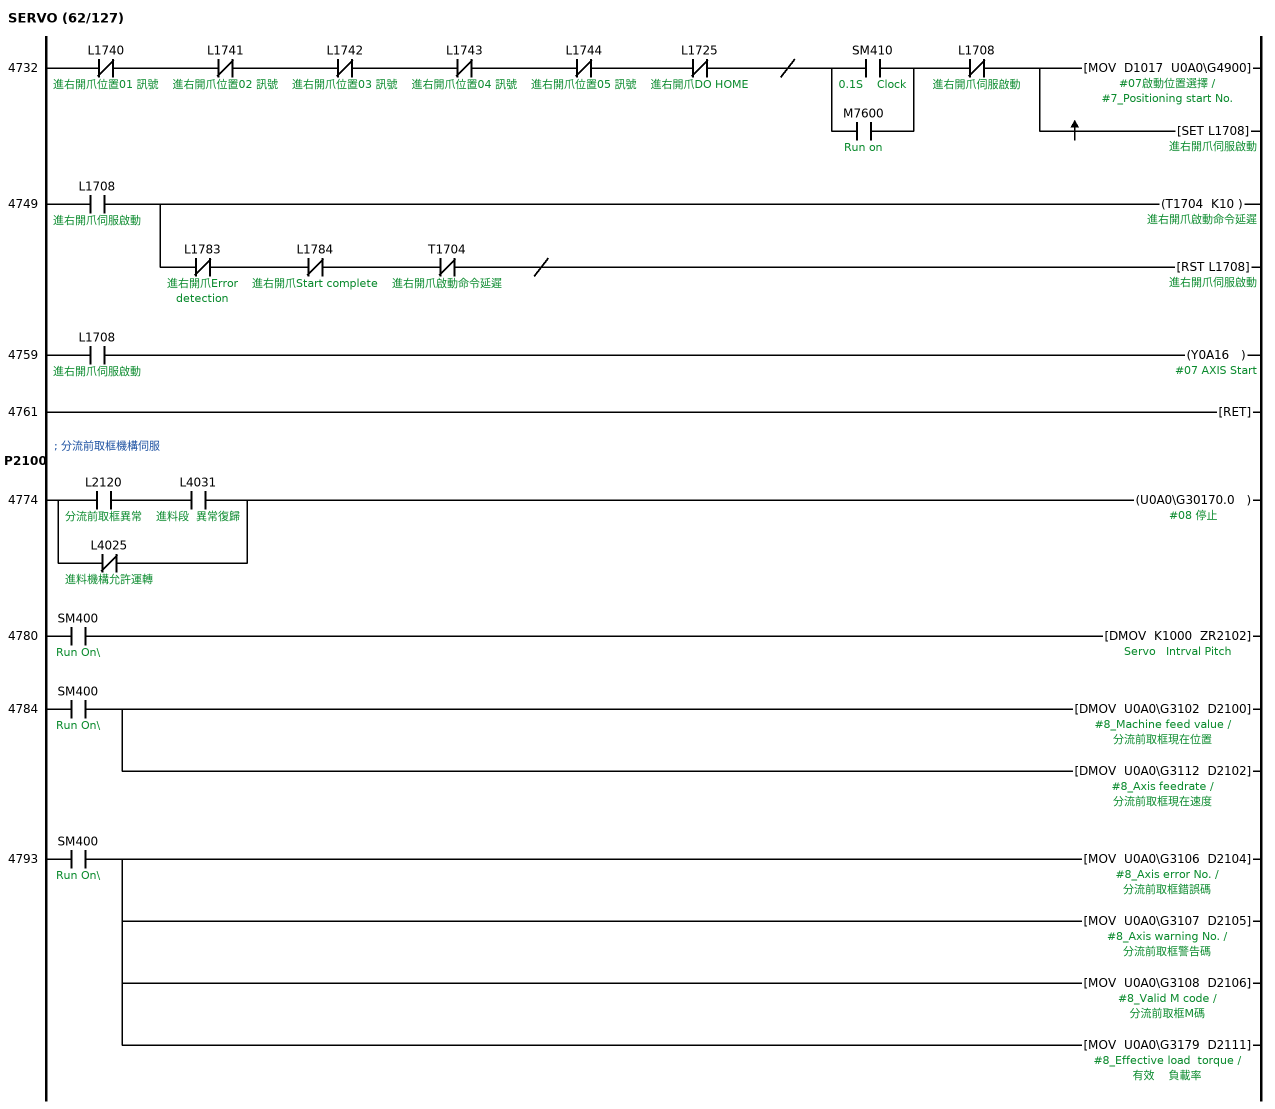
4732  LDI     L1740  ; 進右開爪位置01 訊號
      ANI     L1741  ; 進右開爪位置02 訊號
      ANI     L1742  ; 進右開爪位置03 訊號
      ANI     L1743  ; 進右開爪位置04 訊號
      ANI     L1744  ; 進右開爪位置05 訊號
      ANI     L1725  ; 進右開爪DO HOME
      INV
      LD      SM410  ; 0.1S    Clock
      OR      M7600  ; Run on
      ANB
      ANI     L1708  ; 進右開爪伺服啟動
      MOV     D1017 U0A0\G4900  ; #7_Positioning start No.
      MEP
      SET     L1708  ; 進右開爪伺服啟動
4749  LD      L1708  ; 進右開爪伺服啟動
      OUT     T1704 K10  ; 進右開爪啟動命令延遲
      ANI     L1783  ; 進右開爪Error detection
      ANI     L1784  ; 進右開爪Start complete
      ANI     T1704  ; 進右開爪啟動命令延遲
      INV
      RST     L1708  ; 進右開爪伺服啟動
4759  LD      L1708  ; 進右開爪伺服啟動
      OUT     Y0A16  ; #07 AXIS Start
4761  RET
; 分流前取框機構伺服
      P2100
4774  LD      L2120  ; 分流前取框異常
      AND     L4031  ; 進料段  異常復歸
      ORI     L4025  ; 進料機構允許運轉
      OUT     U0A0\G30170.0  ; #08 停止
4780  LD      SM400  ; Run On\
      DMOV    K1000 ZR2102  ; Servo   Intrval Pitch
4784  LD      SM400  ; Run On\
      DMOV    U0A0\G3102 D2100  ; #8_Machine feed value / 分流前取框現在位置
      DMOV    U0A0\G3112 D2102  ; #8_Axis feedrate / 分流前取框現在速度
4793  LD      SM400  ; Run On\
      MOV     U0A0\G3106 D2104  ; #8_Axis error No. / 分流前取框錯誤碼
      MOV     U0A0\G3107 D2105  ; #8_Axis warning No. / 分流前取框警告碼
      MOV     U0A0\G3108 D2106  ; #8_Valid M code / 分流前取框M碼
      MOV     U0A0\G3179 D2111  ; #8_Effective load  torque / 有效    負載率
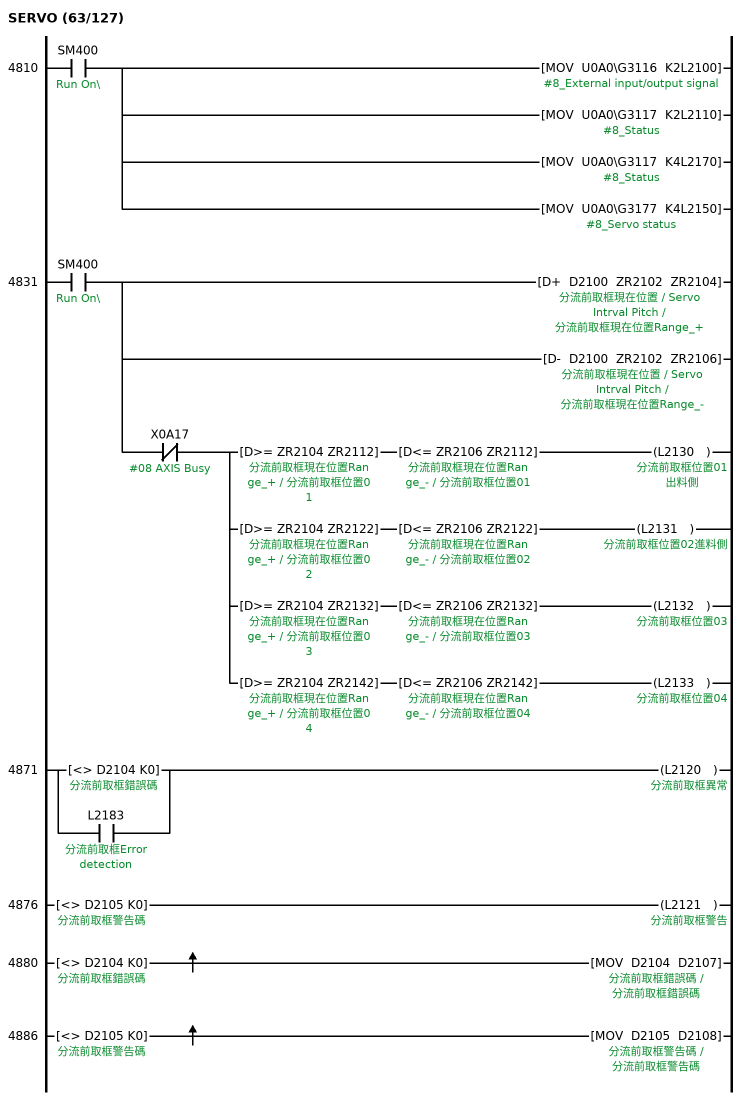
4810  LD      SM400  ; Run On\
      MOV     U0A0\G3116 K2L2100  ; #8_External input/output signal / 分流前取框    負極限
      MOV     U0A0\G3117 K2L2110  ; #8_Status / 分流前取框速度控制
      MOV     U0A0\G3117 K4L2170  ; 分流前取框速度控制
      MOV     U0A0\G3177 K4L2150  ; #8_Servo status / READY ON
4831  LD      SM400  ; Run On\
      D+      D2100 ZR2102 ZR2104  ; 分流前取框現在位置Range_+
      D-      D2100 ZR2102 ZR2106  ; 分流前取框現在位置Range_-
      ANI     X0A17  ; #08 AXIS Busy
      MPS
      ANDD>=  ZR2104 ZR2112  ; 分流前取框現在位置Range_+ / 分流前取框位置01
      ANDD<=  ZR2106 ZR2112  ; 分流前取框現在位置Range_- / 分流前取框位置01
      OUT     L2130  ; 分流前取框位置01  出料側
      MRD
      ANDD>=  ZR2104 ZR2122  ; 分流前取框現在位置Range_+ / 分流前取框位置02
      ANDD<=  ZR2106 ZR2122  ; 分流前取框現在位置Range_- / 分流前取框位置02
      OUT     L2131  ; 分流前取框位置02進料側
      MRD
      ANDD>=  ZR2104 ZR2132  ; 分流前取框現在位置Range_+ / 分流前取框位置03
      ANDD<=  ZR2106 ZR2132  ; 分流前取框現在位置Range_- / 分流前取框位置03
      OUT     L2132  ; 分流前取框位置03
      MPP
      ANDD>=  ZR2104 ZR2142  ; 分流前取框現在位置Range_+ / 分流前取框位置04
      ANDD<=  ZR2106 ZR2142  ; 分流前取框現在位置Range_- / 分流前取框位置04
      OUT     L2133  ; 分流前取框位置04
4871  LD<>    D2104 K0  ; 分流前取框錯誤碼
      OR      L2183  ; 分流前取框Error detection
      OUT     L2120  ; 分流前取框異常
4876  LD<>    D2105 K0  ; 分流前取框警告碼
      OUT     L2121  ; 分流前取框警告
4880  LD<>    D2104 K0  ; 分流前取框錯誤碼
      MEP
      MOV     D2104 D2107  ; 分流前取框錯誤碼
4886  LD<>    D2105 K0  ; 分流前取框警告碼
      MEP
      MOV     D2105 D2108  ; 分流前取框警告碼
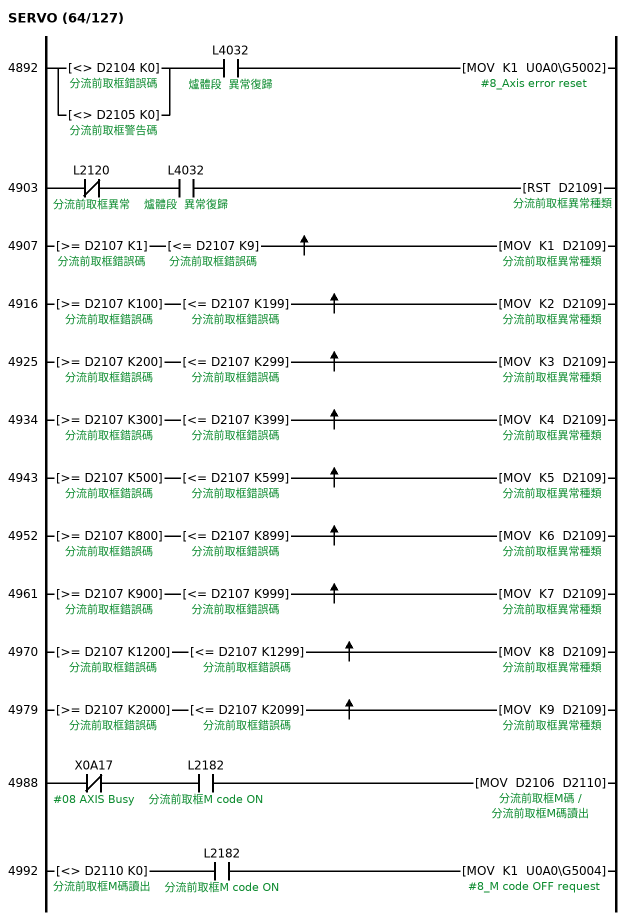
4892  LD<>    D2104 K0  ; 分流前取框錯誤碼
      OR<>    D2105 K0  ; 分流前取框警告碼
      AND     L4032  ; 爐體段  異常復歸
      MOV     K1 U0A0\G5002  ; #8_Axis error reset
4903  LDI     L2120  ; 分流前取框異常
      AND     L4032  ; 爐體段  異常復歸
      RST     D2109  ; 分流前取框異常種類
4907  LD>=    D2107 K1  ; 分流前取框錯誤碼
      AND<=   D2107 K9  ; 分流前取框錯誤碼
      MEP
      MOV     K1 D2109
4916  LD>=    D2107 K100  ; 分流前取框錯誤碼
      AND<=   D2107 K199  ; 分流前取框錯誤碼
      MEP
      MOV     K2 D2109
4925  LD>=    D2107 K200  ; 分流前取框錯誤碼
      AND<=   D2107 K299  ; 分流前取框錯誤碼
      MEP
      MOV     K3 D2109
4934  LD>=    D2107 K300  ; 分流前取框錯誤碼
      AND<=   D2107 K399  ; 分流前取框錯誤碼
      MEP
      MOV     K4 D2109
4943  LD>=    D2107 K500  ; 分流前取框錯誤碼
      AND<=   D2107 K599  ; 分流前取框錯誤碼
      MEP
      MOV     K5 D2109
4952  LD>=    D2107 K800  ; 分流前取框錯誤碼
      AND<=   D2107 K899  ; 分流前取框錯誤碼
      MEP
      MOV     K6 D2109
4961  LD>=    D2107 K900  ; 分流前取框錯誤碼
      AND<=   D2107 K999  ; 分流前取框錯誤碼
      MEP
      MOV     K7 D2109
4970  LD>=    D2107 K1200  ; 分流前取框錯誤碼
      AND<=   D2107 K1299  ; 分流前取框錯誤碼
      MEP
      MOV     K8 D2109
4979  LD>=    D2107 K2000  ; 分流前取框錯誤碼
      AND<=   D2107 K2099  ; 分流前取框錯誤碼
      MEP
      MOV     K9 D2109
4988  LDI     X0A17  ; #08 AXIS Busy
      AND     L2182  ; 分流前取框M code ON
      MOV     D2106 D2110  ; 分流前取框M碼讀出
4992  LD<>    D2110 K0  ; 分流前取框M碼讀出
      AND     L2182  ; 分流前取框M code ON
      MOV     K1 U0A0\G5004  ; #8_M code OFF request
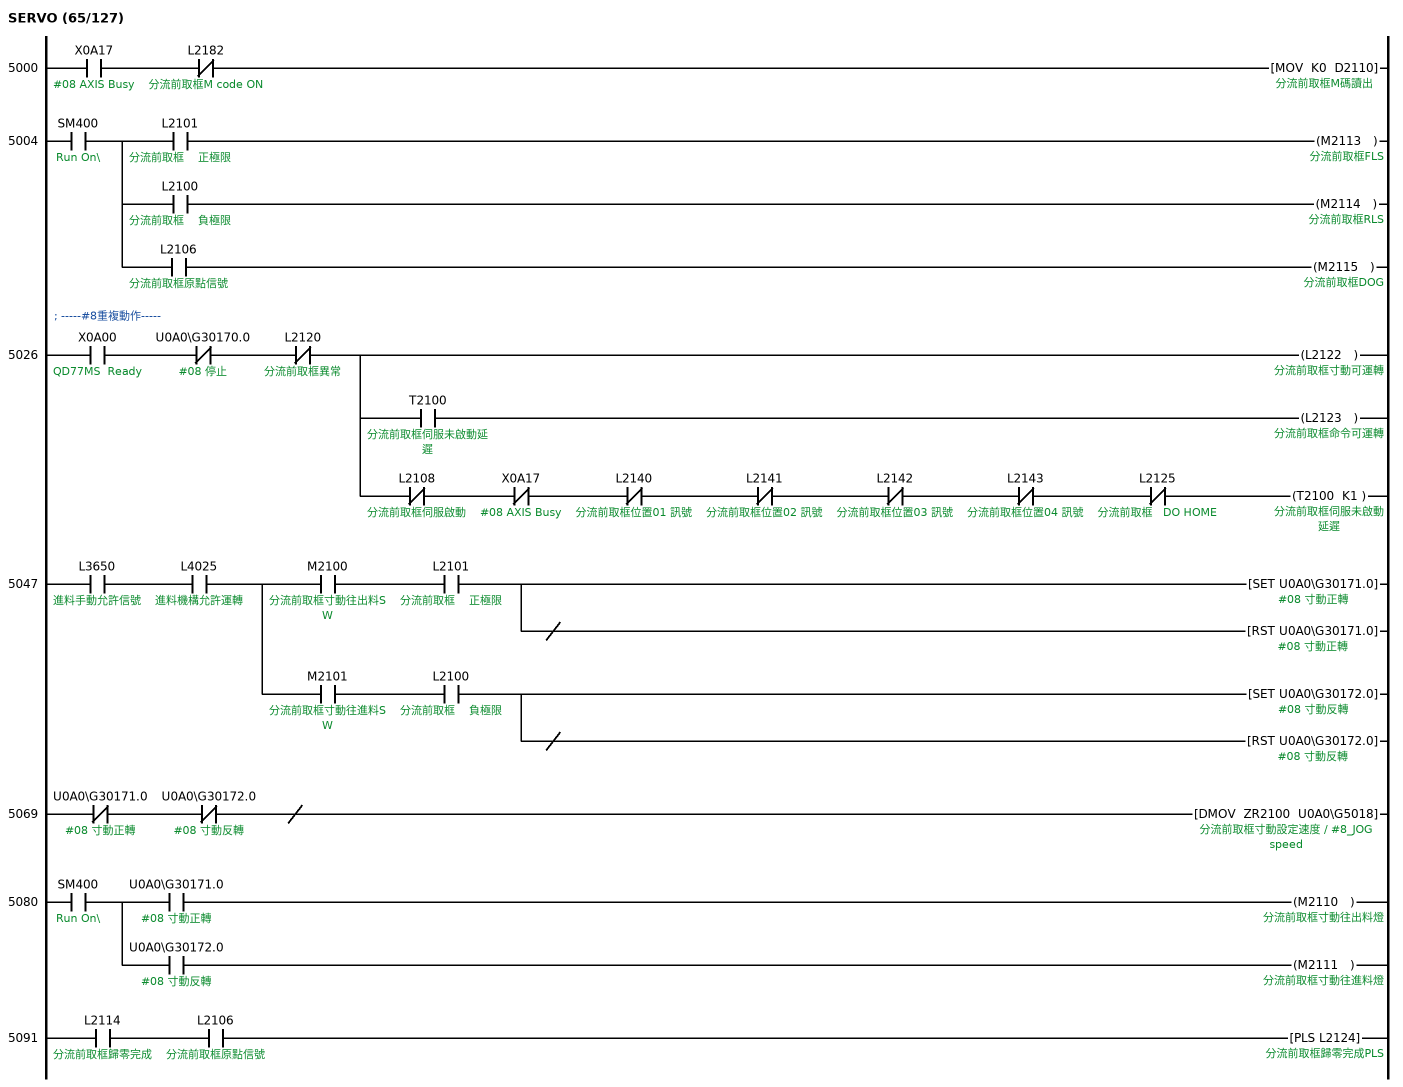
5000  LD      X0A17  ; #08 AXIS Busy
      ANI     L2182  ; 分流前取框M code ON
      MOV     K0 D2110
5004  LD      SM400  ; Run On\
      MPS
      AND     L2101  ; 分流前取框    正極限
      OUT     M2113  ; 分流前取框FLS
      MRD
      AND     L2100  ; 分流前取框    負極限
      OUT     M2114  ; 分流前取框RLS
      MPP
      AND     L2106  ; 分流前取框原點信號
      OUT     M2115  ; 分流前取框DOG
; -----#8重複動作-----
5026  LD      X0A00  ; QD77MS  Ready
      ANI     U0A0\G30170.0  ; #08 停止
      ANI     L2120  ; 分流前取框異常
      OUT     L2122  ; 分流前取框寸動可運轉
      MPS
      AND     T2100  ; 分流前取框伺服未啟動延遲
      OUT     L2123  ; 分流前取框命令可運轉
      MPP
      ANI     L2108  ; 分流前取框伺服啟動
      ANI     X0A17  ; #08 AXIS Busy
      ANI     L2140  ; 分流前取框位置01 訊號
      ANI     L2141  ; 分流前取框位置02 訊號
      ANI     L2142  ; 分流前取框位置03 訊號
      ANI     L2143  ; 分流前取框位置04 訊號
      ANI     L2125  ; 分流前取框   DO HOME
      OUT     T2100 K1  ; 分流前取框伺服未啟動延遲
5047  LD      L3650  ; 進料手動允許信號
      AND     L4025  ; 進料機構允許運轉
      MPS
      AND     M2100  ; 分流前取框寸動往出料SW
      AND     L2101  ; 分流前取框    正極限
      SET     U0A0\G30171.0  ; #08 寸動正轉
      INV
      RST     U0A0\G30171.0  ; #08 寸動正轉
      MPP
      AND     M2101  ; 分流前取框寸動往進料SW
      AND     L2100  ; 分流前取框    負極限
      SET     U0A0\G30172.0  ; #08 寸動反轉
      INV
      RST     U0A0\G30172.0  ; #08 寸動反轉
5069  LDI     U0A0\G30171.0  ; #08 寸動正轉
      ANI     U0A0\G30172.0  ; #08 寸動反轉
      INV
      DMOV    ZR2100 U0A0\G5018  ; 分流前取框寸動設定速度 / #8_JOG     speed
5080  LD      SM400  ; Run On\
      MPS
      AND     U0A0\G30171.0  ; #08 寸動正轉
      OUT     M2110  ; 分流前取框寸動往出料燈
      MPP
      AND     U0A0\G30172.0  ; #08 寸動反轉
      OUT     M2111  ; 分流前取框寸動往進料燈
5091  LD      L2114  ; 分流前取框歸零完成
      AND     L2106  ; 分流前取框原點信號
      PLS     L2124  ; 分流前取框歸零完成PLS
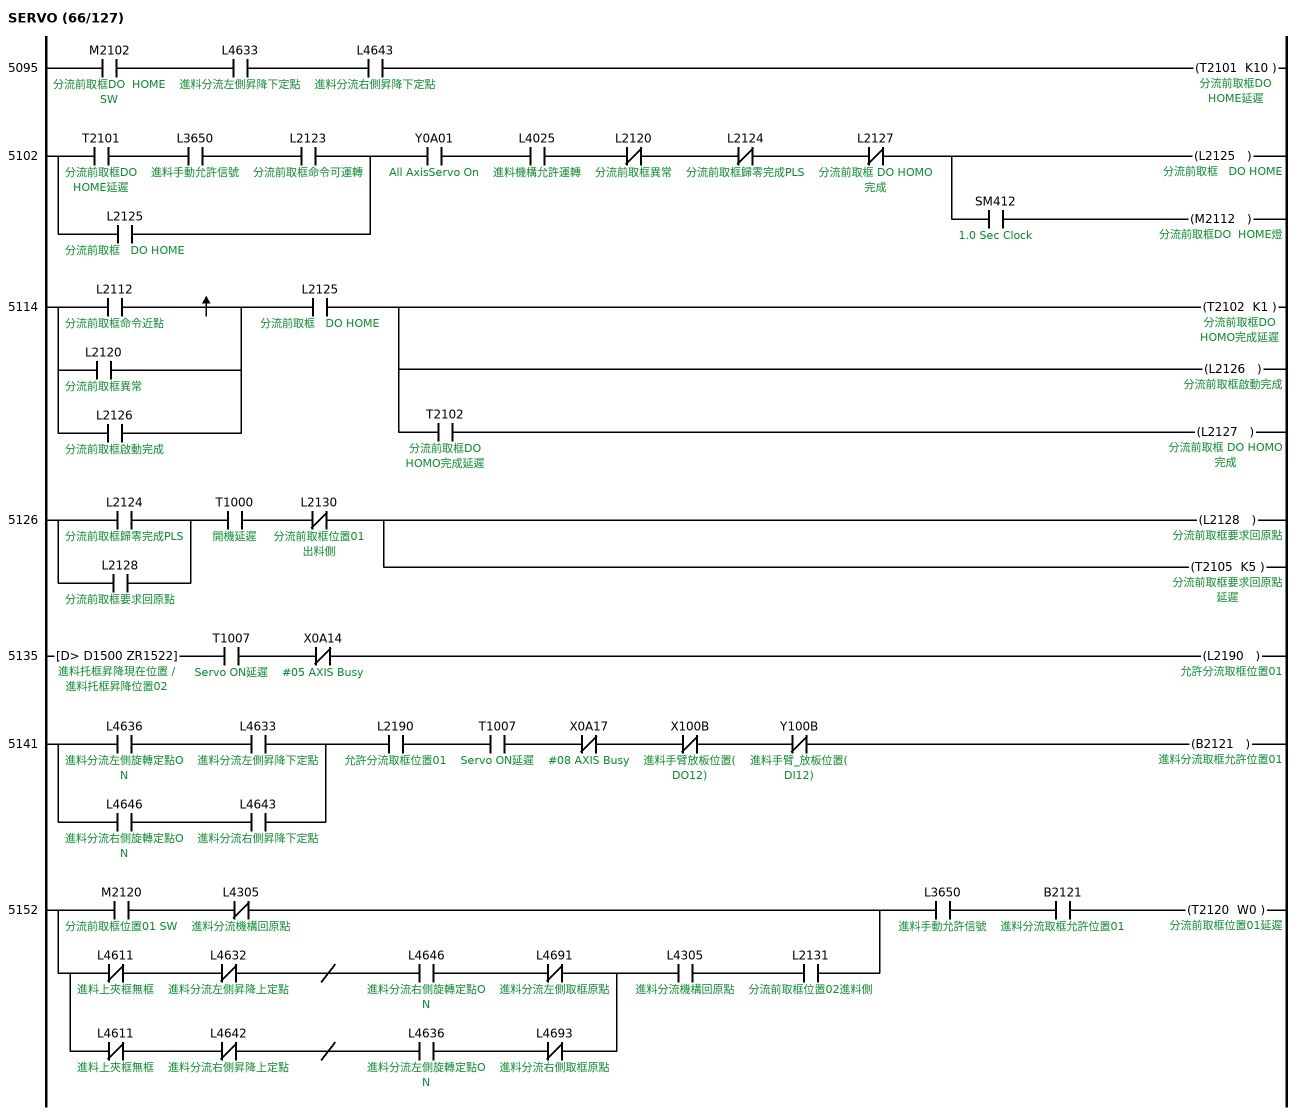
5095  LD      M2102  ; 分流前取框DO  HOME SW
      AND     L4633  ; 進料分流左側昇降下定點
      AND     L4643  ; 進料分流右側昇降下定點
      OUT     T2101 K10  ; 分流前取框DO HOME延遲
5102  LD      T2101  ; 分流前取框DO HOME延遲
      AND     L3650  ; 進料手動允許信號
      AND     L2123  ; 分流前取框命令可運轉
      OR      L2125  ; 分流前取框   DO HOME
      AND     Y0A01  ; All AxisServo On
      AND     L4025  ; 進料機構允許運轉
      ANI     L2120  ; 分流前取框異常
      ANI     L2124  ; 分流前取框歸零完成PLS
      ANI     L2127  ; 分流前取框 DO HOMO 完成
      OUT     L2125  ; 分流前取框   DO HOME
      AND     SM412  ; 1.0 Sec Clock
      OUT     M2112  ; 分流前取框DO  HOME燈
5114  LD      L2112  ; 分流前取框命令近點
      MEP
      OR      L2120  ; 分流前取框異常
      OR      L2126  ; 分流前取框啟動完成
      AND     L2125  ; 分流前取框   DO HOME
      OUT     T2102 K1  ; 分流前取框DO HOMO完成延遲
      OUT     L2126  ; 分流前取框啟動完成
      AND     T2102  ; 分流前取框DO HOMO完成延遲
      OUT     L2127  ; 分流前取框 DO HOMO 完成
5126  LD      L2124  ; 分流前取框歸零完成PLS
      OR      L2128  ; 分流前取框要求回原點
      AND     T1000  ; 開機延遲
      ANI     L2130  ; 分流前取框位置01  出料側
      OUT     L2128  ; 分流前取框要求回原點
      OUT     T2105 K5  ; 分流前取框要求回原點延遲
5135  LDD>    D1500 ZR1522  ; 進料托框昇降現在位置 / 進料托框昇降位置02
      AND     T1007  ; Servo ON延遲
      ANI     X0A14  ; #05 AXIS Busy
      OUT     L2190  ; 允許分流取框位置01
5141  LD      L4636  ; 進料分流左側旋轉定點ON
      AND     L4633  ; 進料分流左側昇降下定點
      LD      L4646  ; 進料分流右側旋轉定點ON
      AND     L4643  ; 進料分流右側昇降下定點
      ORB
      AND     L2190  ; 允許分流取框位置01
      AND     T1007  ; Servo ON延遲
      ANI     X0A17  ; #08 AXIS Busy
      ANI     X100B  ; 進料手臂放板位置(DO12)
      ANI     Y100B  ; 進料手臂_放板位置(DI12)
      OUT     B2121  ; 進料分流取框允許位置01
5152  LD      M2120  ; 分流前取框位置01 SW
      ANI     L4305  ; 進料分流機構回原點
      LDI     L4611  ; 進料上夾框無框
      ANI     L4632  ; 進料分流左側昇降上定點
      INV
      AND     L4646  ; 進料分流右側旋轉定點ON
      ANI     L4691  ; 進料分流左側取框原點
      LDI     L4611  ; 進料上夾框無框
      ANI     L4642  ; 進料分流右側昇降上定點
      INV
      AND     L4636  ; 進料分流左側旋轉定點ON
      ANI     L4693  ; 進料分流右側取框原點
      ORB
      AND     L4305  ; 進料分流機構回原點
      AND     L2131  ; 分流前取框位置02進料側
      ORB
      AND     L3650  ; 進料手動允許信號
      AND     B2121  ; 進料分流取框允許位置01
      OUT     T2120 W0  ; 分流前取框位置01延遲
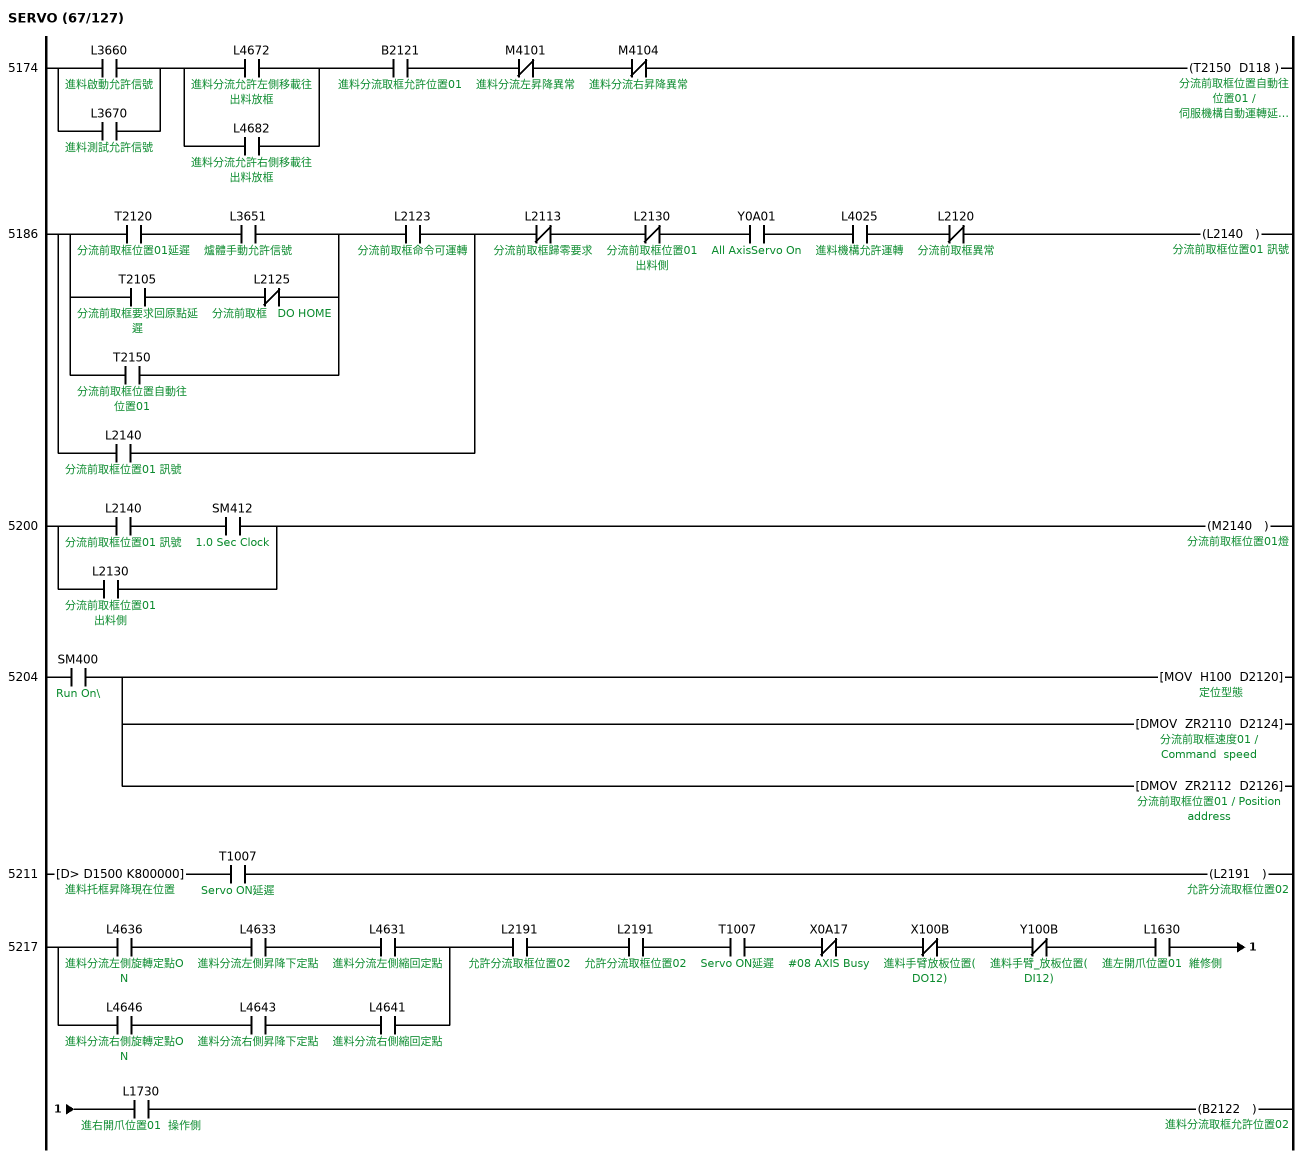
5174  LD      L3660  ; 進料啟動允許信號
      OR      L3670  ; 進料測試允許信號
      LD      L4672  ; 進料分流允許左側移載往  出料放框
      OR      L4682  ; 進料分流允許右側移載往  出料放框
      ANB
      AND     B2121  ; 進料分流取框允許位置01
      ANI     M4101  ; 進料分流左昇降異常
      ANI     M4104  ; 進料分流右昇降異常
      OUT     T2150 D118  ; 分流前取框位置自動往  位置01 / 伺服機構自動運轉延遲時間
5186  LD      T2120  ; 分流前取框位置01延遲
      AND     L3651  ; 爐體手動允許信號
      LD      T2105  ; 分流前取框要求回原點延遲
      ANI     L2125  ; 分流前取框   DO HOME
      ORB
      OR      T2150  ; 分流前取框位置自動往  位置01
      AND     L2123  ; 分流前取框命令可運轉
      OR      L2140  ; 分流前取框位置01 訊號
      ANI     L2113  ; 分流前取框歸零要求
      ANI     L2130  ; 分流前取框位置01  出料側
      AND     Y0A01  ; All AxisServo On
      AND     L4025  ; 進料機構允許運轉
      ANI     L2120  ; 分流前取框異常
      OUT     L2140  ; 分流前取框位置01 訊號
5200  LD      L2140  ; 分流前取框位置01 訊號
      AND     SM412  ; 1.0 Sec Clock
      OR      L2130  ; 分流前取框位置01  出料側
      OUT     M2140  ; 分流前取框位置01燈
5204  LD      SM400  ; Run On\
      MOV     H100 D2120  ; 定位型態
      DMOV    ZR2110 D2124  ; 分流前取框速度01 / Command  speed
      DMOV    ZR2112 D2126  ; Position address
5211  LDD>    D1500 K800000  ; 進料托框昇降現在位置
      AND     T1007  ; Servo ON延遲
      OUT     L2191  ; 允許分流取框位置02
5217  LD      L4636  ; 進料分流左側旋轉定點ON
      AND     L4633  ; 進料分流左側昇降下定點
      AND     L4631  ; 進料分流左側縮回定點
      LD      L4646  ; 進料分流右側旋轉定點ON
      AND     L4643  ; 進料分流右側昇降下定點
      AND     L4641  ; 進料分流右側縮回定點
      ORB
      AND     L2191  ; 允許分流取框位置02
      AND     L2191  ; 允許分流取框位置02
      AND     T1007  ; Servo ON延遲
      ANI     X0A17  ; #08 AXIS Busy
      ANI     X100B  ; 進料手臂放板位置(DO12)
      ANI     Y100B  ; 進料手臂_放板位置(DI12)
      AND     L1630  ; 進左開爪位置01  維修側
      AND     L1730  ; 進右開爪位置01  操作側
      OUT     B2122  ; 進料分流取框允許位置02
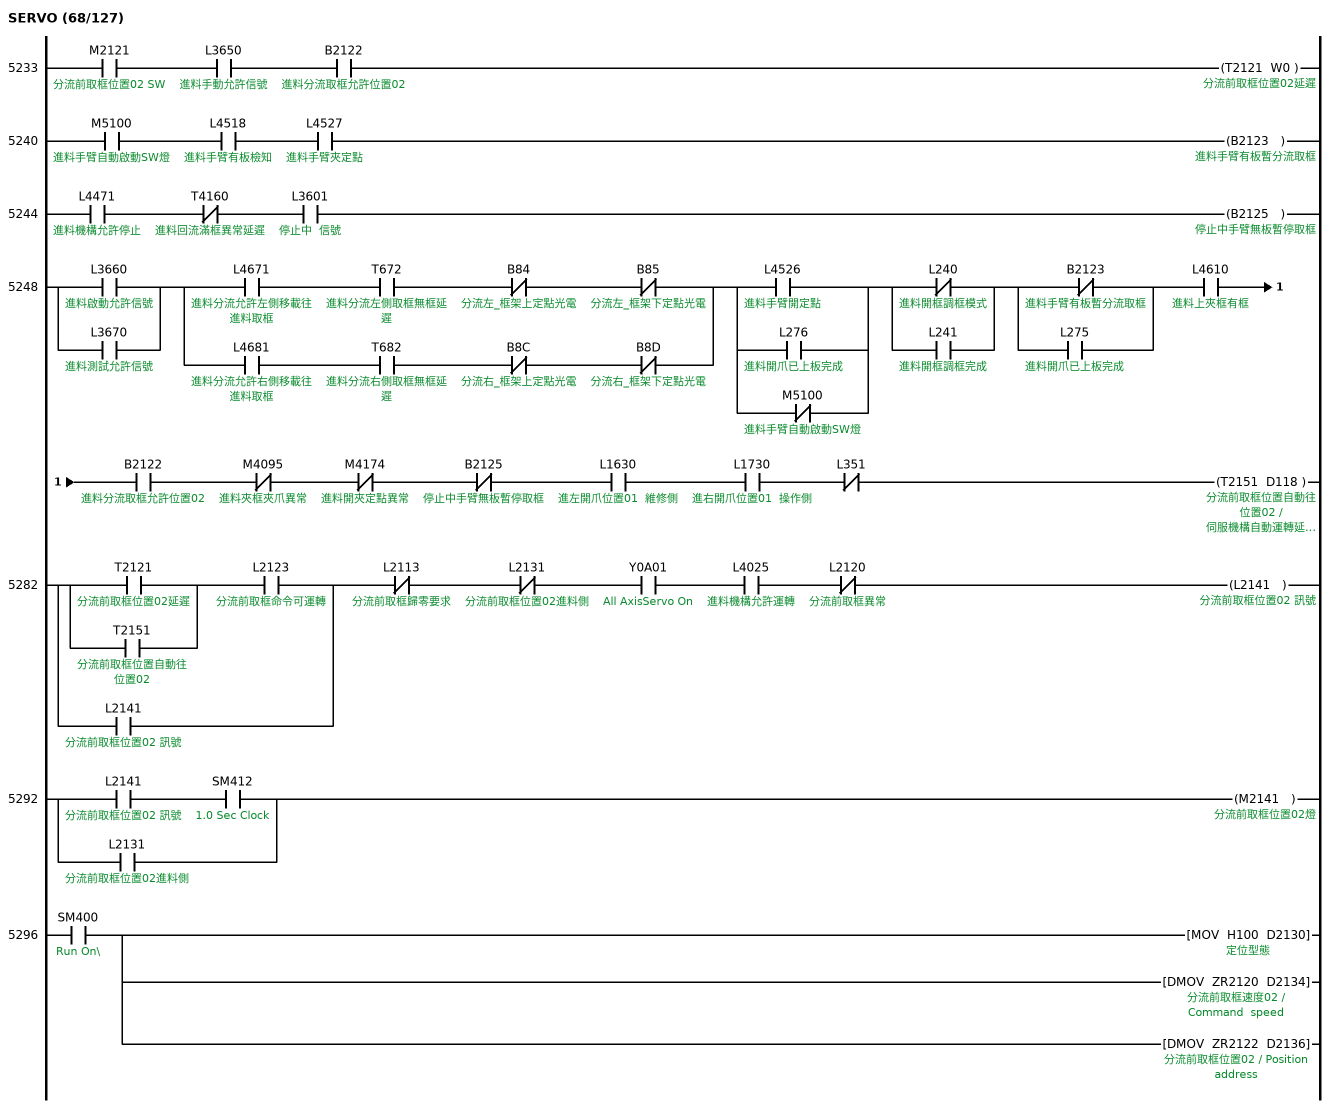
5233  LD      M2121  ; 分流前取框位置02 SW
      AND     L3650  ; 進料手動允許信號
      AND     B2122  ; 進料分流取框允許位置02
      OUT     T2121 W0  ; 分流前取框位置02延遲
5240  LD      M5100  ; 進料手臂自動啟動SW燈
      AND     L4518  ; 進料手臂有板檢知
      AND     L4527  ; 進料手臂夾定點
      OUT     B2123  ; 進料手臂有板暫分流取框
5244  LD      L4471  ; 進料機構允許停止
      ANI     T4160  ; 進料回流滿框異常延遲
      AND     L3601  ; 停止中  信號
      OUT     B2125  ; 停止中手臂無板暫停取框
5248  LD      L3660  ; 進料啟動允許信號
      OR      L3670  ; 進料測試允許信號
      LD      L4671  ; 進料分流允許左側移載往  進料取框
      AND     T672  ; 進料分流左側取框無框延遲
      ANI     B84  ; 分流左_框架上定點光電
      ANI     B85  ; 分流左_框架下定點光電
      LD      L4681  ; 進料分流允許右側移載往  進料取框
      AND     T682  ; 進料分流右側取框無框延遲
      ANI     B8C  ; 分流右_框架上定點光電
      ANI     B8D  ; 分流右_框架下定點光電
      ORB
      ANB
      LD      L4526  ; 進料手臂開定點
      OR      L276  ; 進料開爪已上板完成
      ORI     M5100  ; 進料手臂自動啟動SW燈
      ANB
      LDI     L240  ; 進料開框調框模式
      OR      L241  ; 進料開框調框完成
      ANB
      LDI     B2123  ; 進料手臂有板暫分流取框
      OR      L275  ; 進料開爪已上板完成
      ANB
      AND     L4610  ; 進料上夾框有框
      AND     B2122  ; 進料分流取框允許位置02
      ANI     M4095  ; 進料夾框夾爪異常
      ANI     M4174  ; 進料開夾定點異常
      ANI     B2125  ; 停止中手臂無板暫停取框
      AND     L1630  ; 進左開爪位置01  維修側
      AND     L1730  ; 進右開爪位置01  操作側
      ANI     L351
      OUT     T2151 D118  ; 分流前取框位置自動往  位置02 / 伺服機構自動運轉延遲時間
5282  LD      T2121  ; 分流前取框位置02延遲
      OR      T2151  ; 分流前取框位置自動往  位置02
      AND     L2123  ; 分流前取框命令可運轉
      OR      L2141  ; 分流前取框位置02 訊號
      ANI     L2113  ; 分流前取框歸零要求
      ANI     L2131  ; 分流前取框位置02進料側
      AND     Y0A01  ; All AxisServo On
      AND     L4025  ; 進料機構允許運轉
      ANI     L2120  ; 分流前取框異常
      OUT     L2141  ; 分流前取框位置02 訊號
5292  LD      L2141  ; 分流前取框位置02 訊號
      AND     SM412  ; 1.0 Sec Clock
      OR      L2131  ; 分流前取框位置02進料側
      OUT     M2141  ; 分流前取框位置02燈
5296  LD      SM400  ; Run On\
      MOV     H100 D2130  ; 定位型態
      DMOV    ZR2120 D2134  ; 分流前取框速度02 / Command  speed
      DMOV    ZR2122 D2136  ; Position address
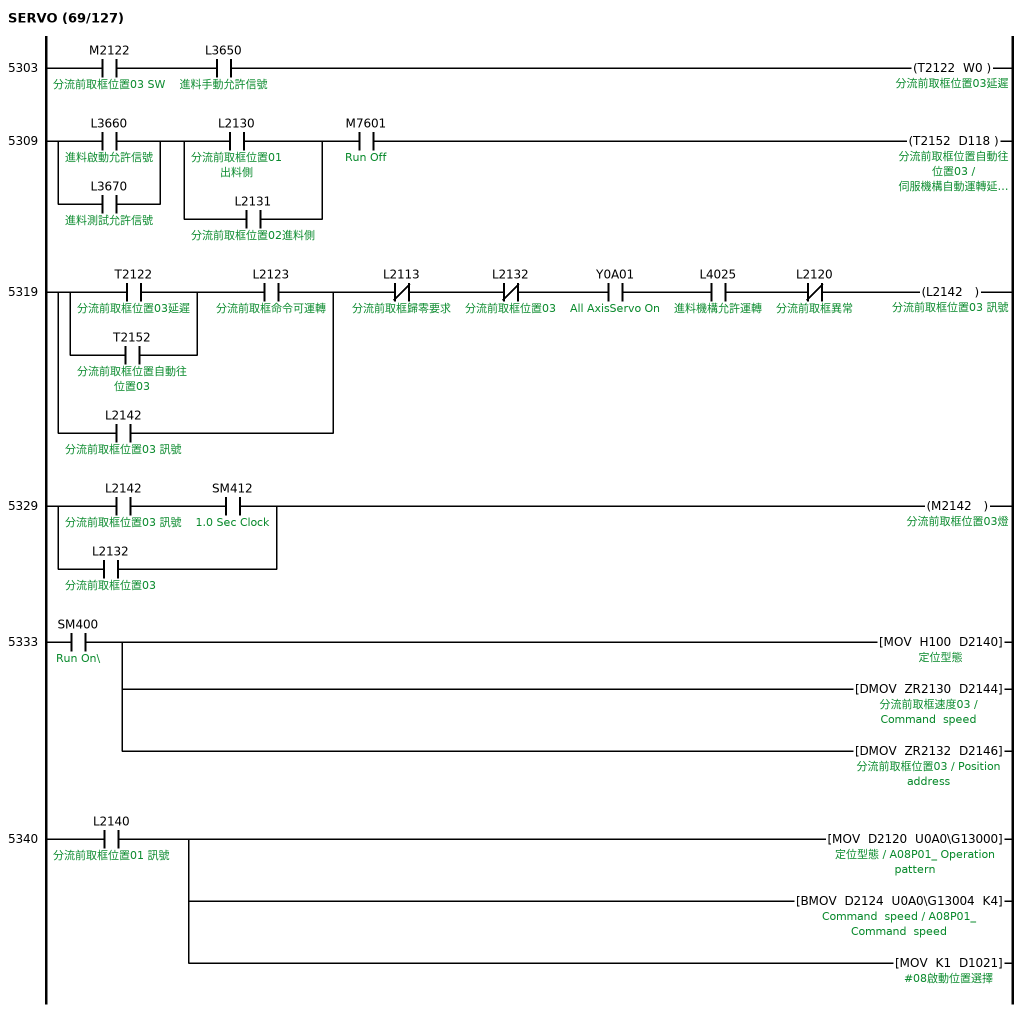
5303  LD      M2122  ; 分流前取框位置03 SW
      AND     L3650  ; 進料手動允許信號
      OUT     T2122 W0  ; 分流前取框位置03延遲
5309  LD      L3660  ; 進料啟動允許信號
      OR      L3670  ; 進料測試允許信號
      LD      L2130  ; 分流前取框位置01  出料側
      OR      L2131  ; 分流前取框位置02進料側
      ANB
      AND     M7601  ; Run Off
      OUT     T2152 D118  ; 分流前取框位置自動往  位置03 / 伺服機構自動運轉延遲時間
5319  LD      T2122  ; 分流前取框位置03延遲
      OR      T2152  ; 分流前取框位置自動往  位置03
      AND     L2123  ; 分流前取框命令可運轉
      OR      L2142  ; 分流前取框位置03 訊號
      ANI     L2113  ; 分流前取框歸零要求
      ANI     L2132  ; 分流前取框位置03
      AND     Y0A01  ; All AxisServo On
      AND     L4025  ; 進料機構允許運轉
      ANI     L2120  ; 分流前取框異常
      OUT     L2142  ; 分流前取框位置03 訊號
5329  LD      L2142  ; 分流前取框位置03 訊號
      AND     SM412  ; 1.0 Sec Clock
      OR      L2132  ; 分流前取框位置03
      OUT     M2142  ; 分流前取框位置03燈
5333  LD      SM400  ; Run On\
      MOV     H100 D2140  ; 定位型態
      DMOV    ZR2130 D2144  ; 分流前取框速度03 / Command  speed
      DMOV    ZR2132 D2146  ; Position address
5340  LD      L2140  ; 分流前取框位置01 訊號
      MOV     D2120 U0A0\G13000  ; A08P01_ Operation pattern
      BMOV    D2124 U0A0\G13004 K4  ; A08P01_ Command  speed
      MOV     K1 D1021  ; #08啟動位置選擇
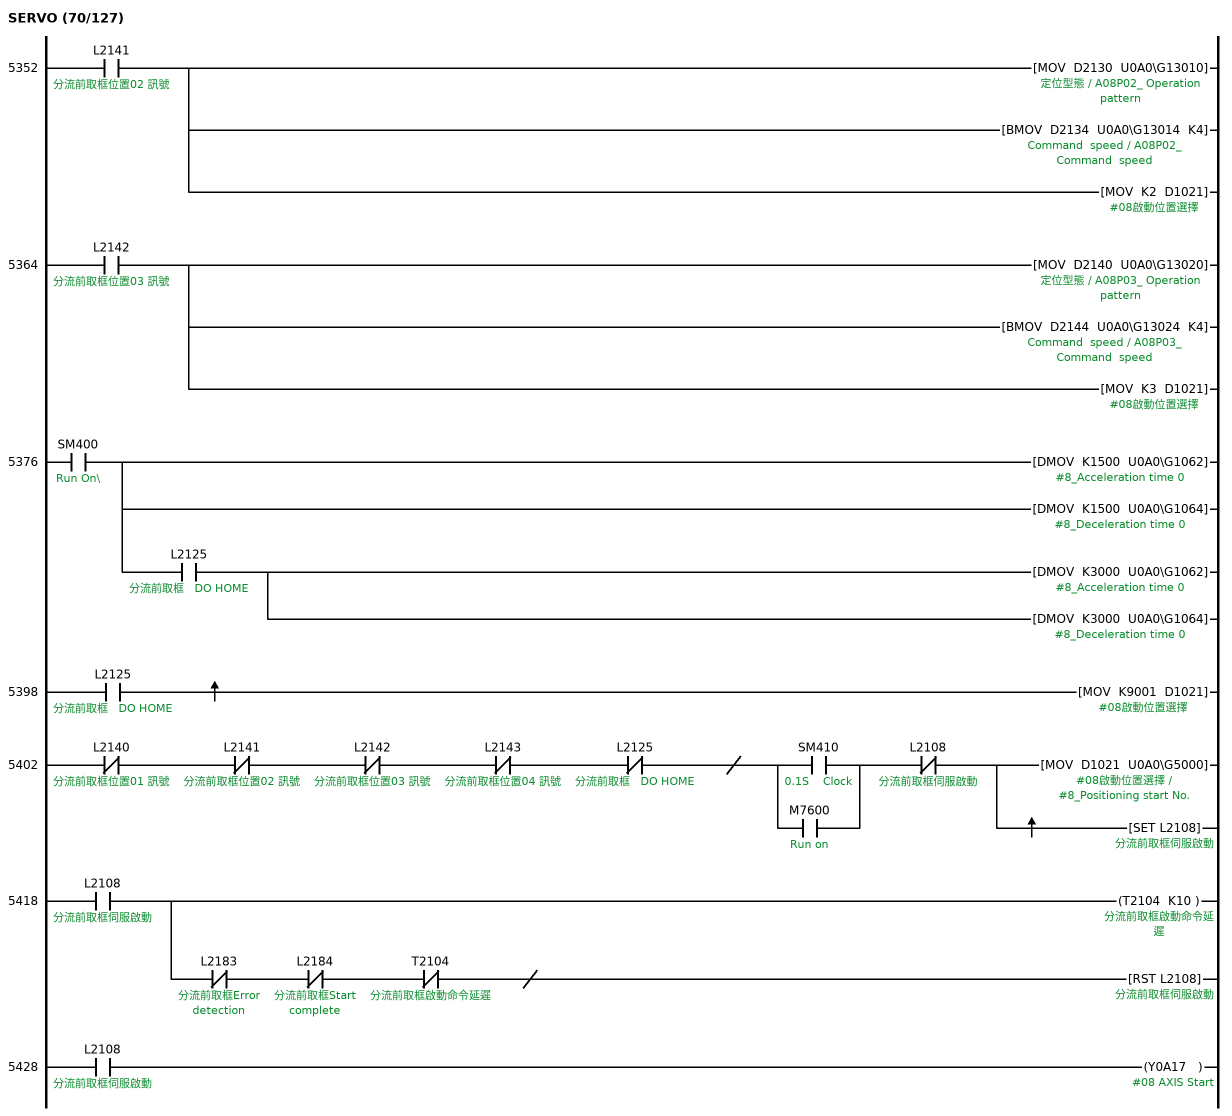
5352  LD      L2141  ; 分流前取框位置02 訊號
      MOV     D2130 U0A0\G13010  ; A08P02_ Operation pattern
      BMOV    D2134 U0A0\G13014 K4  ; A08P02_ Command  speed
      MOV     K2 D1021
5364  LD      L2142  ; 分流前取框位置03 訊號
      MOV     D2140 U0A0\G13020  ; A08P03_ Operation pattern
      BMOV    D2144 U0A0\G13024 K4  ; A08P03_ Command  speed
      MOV     K3 D1021
5376  LD      SM400  ; Run On\
      DMOV    K1500 U0A0\G1062  ; #8_Acceleration time 0
      DMOV    K1500 U0A0\G1064  ; #8_Deceleration time 0
      AND     L2125  ; 分流前取框   DO HOME
      DMOV    K3000 U0A0\G1062
      DMOV    K3000 U0A0\G1064
5398  LD      L2125  ; 分流前取框   DO HOME
      MEP
      MOV     K9001 D1021
5402  LDI     L2140  ; 分流前取框位置01 訊號
      ANI     L2141  ; 分流前取框位置02 訊號
      ANI     L2142  ; 分流前取框位置03 訊號
      ANI     L2143  ; 分流前取框位置04 訊號
      ANI     L2125  ; 分流前取框   DO HOME
      INV
      LD      SM410  ; 0.1S    Clock
      OR      M7600  ; Run on
      ANB
      ANI     L2108  ; 分流前取框伺服啟動
      MOV     D1021 U0A0\G5000  ; #8_Positioning start No.
      MEP
      SET     L2108  ; 分流前取框伺服啟動
5418  LD      L2108  ; 分流前取框伺服啟動
      OUT     T2104 K10  ; 分流前取框啟動命令延遲
      ANI     L2183  ; 分流前取框Error detection
      ANI     L2184  ; 分流前取框Start complete
      ANI     T2104  ; 分流前取框啟動命令延遲
      INV
      RST     L2108  ; 分流前取框伺服啟動
5428  LD      L2108  ; 分流前取框伺服啟動
      OUT     Y0A17  ; #08 AXIS Start
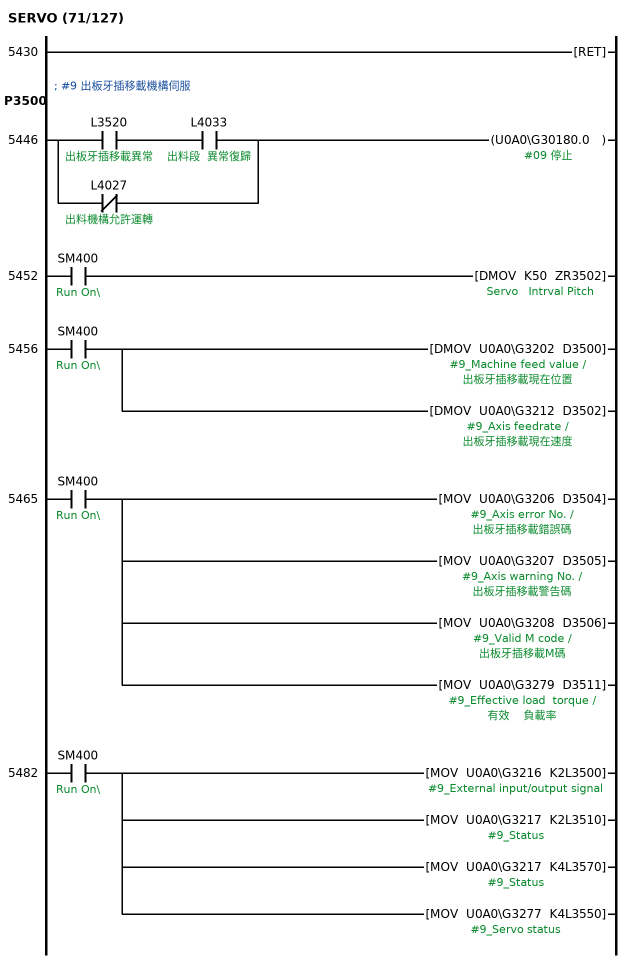
5430  RET
; #9 出板牙插移載機構伺服
      P3500
5446  LD      L3520  ; 出板牙插移載異常
      AND     L4033  ; 出料段  異常復歸
      ORI     L4027  ; 出料機構允許運轉
      OUT     U0A0\G30180.0  ; #09 停止
5452  LD      SM400  ; Run On\
      DMOV    K50 ZR3502  ; Servo   Intrval Pitch
5456  LD      SM400  ; Run On\
      DMOV    U0A0\G3202 D3500  ; #9_Machine feed value / 出板牙插移載現在位置
      DMOV    U0A0\G3212 D3502  ; #9_Axis feedrate / 出板牙插移載現在速度
5465  LD      SM400  ; Run On\
      MOV     U0A0\G3206 D3504  ; #9_Axis error No. / 出板牙插移載錯誤碼
      MOV     U0A0\G3207 D3505  ; #9_Axis warning No. / 出板牙插移載警告碼
      MOV     U0A0\G3208 D3506  ; #9_Valid M code / 出板牙插移載M碼
      MOV     U0A0\G3279 D3511  ; #9_Effective load  torque / 有效    負載率
5482  LD      SM400  ; Run On\
      MOV     U0A0\G3216 K2L3500  ; #9_External input/output signal / 出板牙插移載   負極限
      MOV     U0A0\G3217 K2L3510  ; #9_Status / 出板牙插移載速度控制
      MOV     U0A0\G3217 K4L3570  ; 出板牙插移載速度控制
      MOV     U0A0\G3277 K4L3550  ; #9_Servo status / READY ON
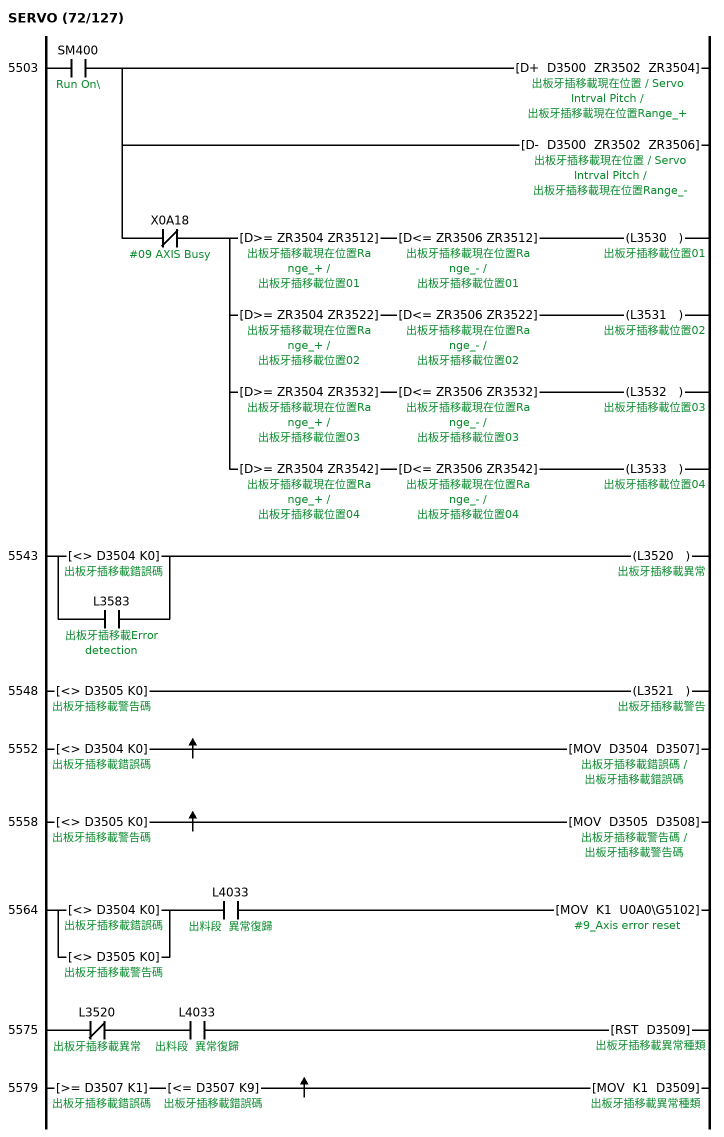
5503  LD      SM400  ; Run On\
      D+      D3500 ZR3502 ZR3504  ; 出板牙插移載現在位置Range_+
      D-      D3500 ZR3502 ZR3506  ; 出板牙插移載現在位置Range_-
      ANI     X0A18  ; #09 AXIS Busy
      MPS
      ANDD>=  ZR3504 ZR3512  ; 出板牙插移載現在位置Range_+ / 出板牙插移載位置01
      ANDD<=  ZR3506 ZR3512  ; 出板牙插移載現在位置Range_- / 出板牙插移載位置01
      OUT     L3530  ; 出板牙插移載位置01
      MRD
      ANDD>=  ZR3504 ZR3522  ; 出板牙插移載現在位置Range_+ / 出板牙插移載位置02
      ANDD<=  ZR3506 ZR3522  ; 出板牙插移載現在位置Range_- / 出板牙插移載位置02
      OUT     L3531  ; 出板牙插移載位置02
      MRD
      ANDD>=  ZR3504 ZR3532  ; 出板牙插移載現在位置Range_+ / 出板牙插移載位置03
      ANDD<=  ZR3506 ZR3532  ; 出板牙插移載現在位置Range_- / 出板牙插移載位置03
      OUT     L3532  ; 出板牙插移載位置03
      MPP
      ANDD>=  ZR3504 ZR3542  ; 出板牙插移載現在位置Range_+ / 出板牙插移載位置04
      ANDD<=  ZR3506 ZR3542  ; 出板牙插移載現在位置Range_- / 出板牙插移載位置04
      OUT     L3533  ; 出板牙插移載位置04
5543  LD<>    D3504 K0  ; 出板牙插移載錯誤碼
      OR      L3583  ; 出板牙插移載Error detection
      OUT     L3520  ; 出板牙插移載異常
5548  LD<>    D3505 K0  ; 出板牙插移載警告碼
      OUT     L3521  ; 出板牙插移載警告
5552  LD<>    D3504 K0  ; 出板牙插移載錯誤碼
      MEP
      MOV     D3504 D3507  ; 出板牙插移載錯誤碼
5558  LD<>    D3505 K0  ; 出板牙插移載警告碼
      MEP
      MOV     D3505 D3508  ; 出板牙插移載警告碼
5564  LD<>    D3504 K0  ; 出板牙插移載錯誤碼
      OR<>    D3505 K0  ; 出板牙插移載警告碼
      AND     L4033  ; 出料段  異常復歸
      MOV     K1 U0A0\G5102  ; #9_Axis error reset
5575  LDI     L3520  ; 出板牙插移載異常
      AND     L4033  ; 出料段  異常復歸
      RST     D3509  ; 出板牙插移載異常種類
5579  LD>=    D3507 K1  ; 出板牙插移載錯誤碼
      AND<=   D3507 K9  ; 出板牙插移載錯誤碼
      MEP
      MOV     K1 D3509
